KUKA KRL program: MyProgram_239().src

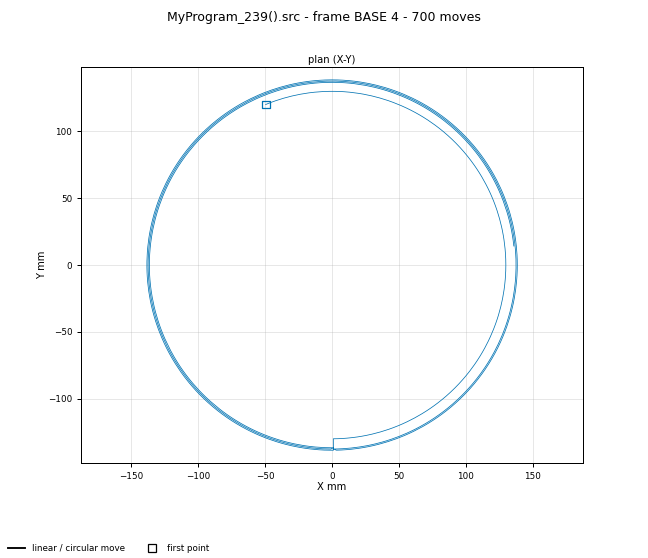
[picture p0: tool path of MyProgram_239().src in frame BASE 4, 700 of 700 moves have a stored position in this frame; points joined in program order, loops and branches not executed]
&ACCESS RVP
&REL 1
&PARAM TEMPLATE = C:\KRC\Roboter\Template\vorgabe
&PARAM EDITMASK = *
DEF MyProgram_239()
; ---- Setting reference (Base) ----
$BASE = BASE_DATA[4]

; --------------------------
; ---- Setting tool (TCP) ----
$TOOL = TOOL_DATA[3]
; --------------------------

$VEL.CP = VEL_APROX_PRINT
Startdeposition()
$VEL.CP = VEL_PRINT
LIN {X -49.7032,Y 120.0061,Z 160,A 111.2749,B 14.0881,C -0.1993,E1 14.0298,E2 338.4805} C_DIS
LIN {X -45.6946,Y 121.5885,Z 160,A 109.4151,B 14.0881,C -0.2026,E1 14.0346,E2 340.334} C_DIS
LIN {X -42.2336,Y 122.834,Z 160,A 107.7853,B 14.0881,C -0.2041,E1 14.0389,E2 341.9633} C_DIS
LIN {X -39.2151,Y 123.8307,Z 160,A 106.3787,B 14.0881,C -0.2054,E1 14.0427,E2 343.3693} C_DIS
LIN {X -36.1716,Y 124.7537,Z 160,A 104.9717,B 14.088,C -0.2066,E1 14.0464,E2 344.7756} C_DIS
LIN {X -33.1062,Y 125.6021,Z 160,A 103.5625,B 14.088,C -0.2076,E1 14.0502,E2 346.1844} C_DIS
LIN {X -29.9974,Y 126.381,Z 160,A 102.1496,B 14.088,C -0.2088,E1 14.0541,E2 347.5962} C_DIS
LIN {X -26.9022,Y 127.0761,Z 160,A 100.7679,B 14.088,C -0.2103,E1 14.0578,E2 348.9749} C_DIS
LIN {X -23.6832,Y 127.7162,Z 160,A 99.3021,B 14.088,C -0.2107,E1 14.0618,E2 350.4419} C_DIS
LIN {X -21.0729,Y 128.1711,Z 160,A 98.0756,B 14.088,C -0.2098,E1 14.0652,E2 351.6741} C_DIS
LIN {X -17.5361,Y 128.7041,Z 160,A 96.3923,B 14.088,C -0.2077,E1 14.0699,E2 353.3685} C_DIS
LIN {X -13.1972,Y 129.2214,Z 160,A 94.4723,B 14.088,C -0.2087,E1 14.0752,E2 355.2865} C_DIS
LIN {X -9.5576,Y 129.5396,Z 160,A 92.993,B 14.088,C -0.2129,E1 14.0793,E2 356.7497} C_DIS
LIN {X -6.3664,Y 129.7357,Z 160,A 91.5337,B 14.088,C -0.2119,E1 14.0834,E2 358.2139} C_DIS
LIN {X -2.0579,Y 129.8755,Z 160,A 89.6356,B 14.088,C -0.2123,E1 14.0887,E2 360.1106} C_DIS
LIN {X 2.062,Y 129.8755,Z 160,A 87.7741,B 14.088,C -0.2112,E1 14.0939,E2 361.9764} C_DIS
LIN {X 5.2462,Y 129.7859,Z 160,A 86.3414,B 14.088,C -0.2104,E1 14.0979,E2 363.4116} C_DIS
LIN {X 9.0939,Y 129.5735,Z 160,A 84.7482,B 14.0879,C -0.2132,E1 14.1023,E2 364.9919} C_DIS
LIN {X 13.1987,Y 129.2212,Z 160,A 82.7681,B 14.0879,C -0.2083,E1 14.1079,E2 366.9899} C_DIS
LIN {X 17.4787,Y 128.7116,Z 160,A 81.0931,B 14.0879,C -0.2141,E1 14.1124,E2 368.6386} C_DIS
LIN {X 20.1102,Y 128.3256,Z 160,A 79.7906,B 14.0879,C -0.21,E1 14.1161,E2 369.9554} C_DIS
LIN {X 23.3548,Y 127.7755,Z 160,A 78.4283,B 14.0879,C -0.2119,E1 14.1198,E2 371.3071} C_DIS
LIN {X 26.9191,Y 127.0724,Z 160,A 76.937,B 14.0879,C -0.2142,E1 14.1238,E2 372.7854} C_DIS
LIN {X 29.569,Y 126.4828,Z 160,A 75.6327,B 14.0879,C -0.2105,E1 14.1274,E2 374.1017} C_DIS
LIN {X 32.6519,Y 125.7225,Z 160,A 74.2354,B 14.0879,C -0.2097,E1 14.1312,E2 375.4984} C_DIS
LIN {X 35.7407,Y 124.8799,Z 160,A 72.8179,B 14.0879,C -0.2085,E1 14.135,E2 376.9163} C_DIS
LIN {X 38.7913,Y 123.9661,Z 160,A 71.4198,B 14.0879,C -0.2076,E1 14.1387,E2 378.3136} C_DIS
LIN {X 41.8166,Y 122.9786,Z 160,A 69.7915,B 14.0881,C -0.1999,E1 14.1431,E2 379.9674} C_DIS
LIN {X 45.6939,Y 121.5888,Z 160,A 68.1327,B 14.0881,C -0.2027,E1 14.1474,E2 381.608} C_DIS
LIN {X 49.2665,Y 120.1879,Z 160,A 66.5276,B 14.0881,C -0.2035,E1 14.1516,E2 383.2031} C_DIS
LIN {X 51.7426,Y 119.1406,Z 160,A 65.2806,B 14.0881,C -0.2004,E1 14.1548,E2 384.4571} C_DIS
LIN {X 55.5451,Y 117.4168,Z 160,A 63.5143,B 14.0881,C -0.2004,E1 14.1592,E2 386.2149} C_DIS
LIN {X 58.8237,Y 115.8081,Z 160,A 61.8469,B 14.0881,C -0.1968,E1 14.1634,E2 387.8889} C_DIS
LIN {X 62.2203,Y 114.0214,Z 160,A 60.1436,B 14.0881,C -0.1942,E1 14.1676,E2 389.5937} C_DIS
LIN {X 65.3999,Y 112.2284,Z 160,A 58.6138,B 14.0881,C -0.1942,E1 14.1713,E2 391.1146} C_DIS
LIN {X 68.1296,Y 110.5923,Z 160,A 57.1082,B 14.0882,C -0.1892,E1 14.1749,E2 392.6322} C_DIS
LIN {X 71.7854,Y 108.2555,Z 160,A 55.3158,B 14.0882,C -0.1898,E1 14.1791,E2 394.4111} C_DIS
LIN {X 74.4134,Y 106.4657,Z 160,A 53.9209,B 14.0882,C -0.1878,E1 14.1823,E2 395.8055} C_DIS
LIN {X 77.0015,Y 104.6089,Z 160,A 52.4462,B 14.0883,C -0.1833,E1 14.1856,E2 397.2886} C_DIS
LIN {X 80.232,Y 102.1521,Z 160,A 50.645,B 14.0883,C -0.1798,E1 14.1896,E2 399.0918} C_DIS
LIN {X 83.2585,Y 99.7013,Z 160,A 48.9085,B 14.0884,C -0.1761,E1 14.1934,E2 400.8311} C_DIS
LIN {X 86.6409,Y 96.7759,Z 160,A 46.989,B 14.0884,C -0.174,E1 14.1974,E2 402.7452} C_DIS
LIN {X 89.734,Y 93.9151,Z 160,A 45.1415,B 14.0884,C -0.1706,E1 14.2012,E2 404.5923} C_DIS
LIN {X 92.613,Y 91.0774,Z 160,A 43.3362,B 14.0885,C -0.1663,E1 14.2047,E2 406.4011} C_DIS
LIN {X 95.7938,Y 87.7259,Z 160,A 41.3052,B 14.0885,C -0.1622,E1 14.2086,E2 408.4323} C_DIS
LIN {X 98.5161,Y 84.6572,Z 160,A 39.5451,B 14.0885,C -0.1597,E1 14.2118,E2 410.1878} C_DIS
LIN {X 101.2684,Y 81.345,Z 160,A 37.6742,B 14.0886,C -0.1563,E1 14.2151,E2 412.0566} C_DIS
LIN {X 103.9483,Y 77.8918,Z 160,A 35.7201,B 14.0886,C -0.151,E1 14.2184,E2 414.0149} C_DIS
LIN {X 106.1955,Y 74.7981,Z 160,A 34.1837,B 14.0886,C -0.1516,E1 14.2209,E2 415.535} C_DIS
LIN {X 107.9969,Y 72.1728,Z 160,A 32.7951,B 14.0887,C -0.1487,E1 14.2231,E2 416.9228} C_DIS
LIN {X 109.9996,Y 69.0825,Z 160,A 31.0479,B 14.0887,C -0.1409,E1 14.2257,E2 418.6855} C_DIS
LIN {X 111.9911,Y 65.8044,Z 160,A 29.5076,B 14.0887,C -0.1413,E1 14.2279,E2 420.2095} C_DIS
LIN {X 113.5692,Y 63.0419,Z 160,A 28.0941,B 14.0888,C -0.1374,E1 14.2299,E2 421.6253} C_DIS
LIN {X 115.0779,Y 60.2396,Z 160,A 26.7243,B 14.0888,C -0.1348,E1 14.2316,E2 422.9922} C_DIS
LIN {X 116.5193,Y 57.402,Z 160,A 25.3351,B 14.0888,C -0.1316,E1 14.2334,E2 424.3809} C_DIS
LIN {X 118.088,Y 54.1033,Z 160,A 23.7352,B 14.0889,C -0.1276,E1 14.2353,E2 425.981} C_DIS
LIN {X 119.3878,Y 51.1708,Z 160,A 22.3362,B 14.0889,C -0.1243,E1 14.2368,E2 427.3793} C_DIS
LIN {X 120.7817,Y 47.7926,Z 160,A 20.6564,B 14.0889,C -0.1177,E1 14.2386,E2 429.0686} C_DIS
LIN {X 122.1392,Y 44.2018,Z 160,A 18.978,B 14.089,C -0.1135,E1 14.2402,E2 430.7468} C_DIS
LIN {X 123.3413,Y 40.7281,Z 160,A 17.4623,B 14.089,C -0.1123,E1 14.2416,E2 432.2517} C_DIS
LIN {X 124.3013,Y 37.697,Z 160,A 16.0749,B 14.089,C -0.1088,E1 14.2427,E2 433.6387} C_DIS
LIN {X 125.187,Y 34.6425,Z 160,A 14.6877,B 14.089,C -0.1052,E1 14.2438,E2 435.0256} C_DIS
LIN {X 125.9978,Y 31.5675,Z 160,A 13.3007,B 14.0891,C -0.1017,E1 14.2447,E2 436.4121} C_DIS
LIN {X 126.7327,Y 28.4748,Z 160,A 11.9153,B 14.0891,C -0.0982,E1 14.2456,E2 437.7971} C_DIS
LIN {X 127.2976,Y 25.829,Z 160,A 10.7066,B 14.0891,C -0.0942,E1 14.2463,E2 439.0088} C_DIS
LIN {X 127.9907,Y 22.1528,Z 160,A 9.1132,B 14.0891,C -0.0911,E1 14.2471,E2 440.5974} C_DIS
LIN {X 128.4876,Y 19.0587,Z 160,A 7.716,B 14.0892,C -0.0866,E1 14.2477,E2 441.9979} C_DIS
LIN {X 128.9711,Y 15.4368,Z 160,A 6.049,B 14.0892,C -0.0801,E1 14.2483,E2 443.6731} C_DIS
LIN {X 129.3109,Y 12.2699,Z 160,A 4.6342,B 14.0892,C -0.0756,E1 14.2487,E2 445.0907} C_DIS
LIN {X 129.6473,Y 7.9637,Z 160,A 2.8627,B 14.0892,C -0.0741,E1 14.249,E2 446.8487} C_DIS
LIN {X 129.822,Y 4.3136,Z 160,A 1.0954,B 14.0893,C -0.0644,E1 14.2492,E2 448.636} C_DIS
LIN {X 129.895,Y 0.007,Z 160,A -0.785,B 14.0893,C -0.0593,E1 14.2492,E2 450.5165} C_DIS
LIN {X 129.822,Y -4.3151,Z 160,A -2.4696,B 14.0893,C -0.0606,E1 14.2492,E2 452.1773} C_DIS
LIN {X 129.676,Y -7.498,Z 160,A -3.9032,B 14.0893,C -0.0555,E1 14.249,E2 453.6158} C_DIS
LIN {X 129.4525,Y -10.6747,Z 160,A -5.4288,B 14.0894,C -0.0475,E1 14.2486,E2 455.1574} C_DIS
LIN {X 128.9724,Y -15.4254,Z 160,A -7.4213,B 14.0894,C -0.0448,E1 14.248,E2 457.1391} C_DIS
LIN {X 128.5535,Y -18.5974,Z 160,A -8.7549,B 14.0894,C -0.043,E1 14.2475,E2 458.4653} C_DIS
LIN {X 127.9752,Y -22.2393,Z 160,A -10.3122,B 14.0894,C -0.0403,E1 14.2468,E2 460.0166} C_DIS
LIN {X 127.4877,Y -24.8786,Z 160,A -11.6353,B 14.0894,C -0.0324,E1 14.2461,E2 461.3574} C_DIS
LIN {X 126.8347,Y -28.0205,Z 160,A -12.933,B 14.0894,C -0.0319,E1 14.2454,E2 462.6432} C_DIS
LIN {X 126.1505,Y -30.9533,Z 160,A -14.2383,B 14.0894,C -0.0288,E1 14.2445,E2 463.9474} C_DIS
LIN {X 125.3166,Y -34.1769,Z 160,A -15.7036,B 14.0894,C -0.0246,E1 14.2435,E2 465.4142} C_DIS
LIN {X 124.433,Y -37.2667,Z 160,A -17.1097,B 14.0894,C -0.0208,E1 14.2424,E2 466.8207} C_DIS
LIN {X 123.4826,Y -40.3039,Z 160,A -18.4978,B 14.0894,C -0.0172,E1 14.2412,E2 468.2088} C_DIS
LIN {X 122.2991,Y -43.7581,Z 160,A -20.2163,B 14.0894,C -0.0092,E1 14.2396,E2 469.942} C_DIS
LIN {X 120.7401,Y -47.8966,Z 160,A -22.0062,B 14.0894,C -0.0087,E1 14.2378,E2 471.7155} C_DIS
LIN {X 119.5532,Y -50.7878,Z 160,A -23.3927,B 14.0894,C -0.0046,E1 14.2363,E2 473.1047} C_DIS
LIN {X 118.3107,Y -53.6163,Z 160,A -24.7448,B 14.0894,C -0.0011,E1 14.2348,E2 474.4573} C_DIS
LIN {X 116.7283,Y -56.9782,Z 160,A -26.352,B 14.0894,C 0.0024,E1 14.2328,E2 476.0628} C_DIS
LIN {X 115.2981,Y -59.8203,Z 160,A -27.7239,B 14.0894,C 0.0053,E1 14.2311,E2 477.4328} C_DIS
LIN {X 114.1159,Y -62.047,Z 160,A -28.9697,B 14.0894,C 0.0125,E1 14.2294,E2 478.6958} C_DIS
LIN {X 112.4647,Y -64.9918,Z 160,A -30.4091,B 14.0894,C 0.0149,E1 14.2274,E2 480.1312} C_DIS
LIN {X 110.5875,Y -68.1374,Z 160,A -31.9279,B 14.0894,C 0.0161,E1 14.2252,E2 481.6406} C_DIS
LIN {X 108.5876,Y -71.2811,Z 160,A -33.662,B 14.0894,C 0.0232,E1 14.2226,E2 483.3874} C_DIS
LIN {X 106.4641,Y -74.4157,Z 160,A -35.2113,B 14.0894,C 0.0237,E1 14.2202,E2 484.9246} C_DIS
LIN {X 104.6112,Y -76.9983,Z 160,A -36.5974,B 14.0894,C 0.0267,E1 14.2179,E2 486.3106} C_DIS
LIN {X 102.8556,Y -79.3288,Z 160,A -38.0201,B 14.0894,C 0.0341,E1 14.2155,E2 487.7509} C_DIS
LIN {X 100.2422,Y -82.6064,Z 160,A -39.8187,B 14.0894,C 0.037,E1 14.2123,E2 489.5459} C_DIS
LIN {X 97.4592,Y -85.8719,Z 160,A -41.6299,B 14.0894,C 0.039,E1 14.209,E2 491.3497} C_DIS
LIN {X 94.7928,Y -88.8071,Z 160,A -43.3846,B 14.0894,C 0.0431,E1 14.2057,E2 493.1072} C_DIS
LIN {X 91.8229,Y -91.8745,Z 160,A -45.341,B 14.0894,C 0.0496,E1 14.2018,E2 495.0744} C_DIS
LIN {X 88.5345,Y -95.0467,Z 160,A -47.2615,B 14.0894,C 0.0511,E1 14.198,E2 496.9861} C_DIS
LIN {X 85.452,Y -97.8273,Z 160,A -49.0529,B 14.0894,C 0.0537,E1 14.1942,E2 498.7749} C_DIS
LIN {X 82.3877,Y -100.4219,Z 160,A -50.8685,B 14.0894,C 0.0586,E1 14.1903,E2 500.5977} C_DIS
LIN {X 79.231,Y -102.9313,Z 160,A -52.6764,B 14.0894,C 0.063,E1 14.1863,E2 502.4111} C_DIS
LIN {X 76.4378,Y -105.0217,Z 160,A -54.1414,B 14.0894,C 0.0637,E1 14.183,E2 503.869} C_DIS
LIN {X 73.4926,Y -107.1031,Z 160,A -55.6315,B 14.0894,C 0.0635,E1 14.1796,E2 505.3489} C_DIS
LIN {X 70.8271,Y -108.8842,Z 160,A -57.1232,B 14.0894,C 0.0684,E1 14.1761,E2 506.8514} C_DIS
LIN {X 67.1774,Y -111.173,Z 160,A -58.9257,B 14.0894,C 0.0686,E1 14.1719,E2 508.6442} C_DIS
LIN {X 64.4349,Y -112.7847,Z 160,A -60.3238,B 14.0894,C 0.0708,E1 14.1685,E2 510.0432} C_DIS
LIN {X 61.7406,Y -114.2822,Z 160,A -61.7623,B 14.0893,C 0.0753,E1 14.165,E2 511.4923} C_DIS
LIN {X 58.8215,Y -115.8091,Z 160,A -63.1186,B 14.0893,C 0.0745,E1 14.1616,E2 512.8385} C_DIS
LIN {X 55.9699,Y -117.2139,Z 160,A -64.5849,B 14.0893,C 0.0785,E1 14.1579,E2 514.3138} C_DIS
LIN {X 52.6245,Y -118.7543,Z 160,A -66.1324,B 14.0893,C 0.0784,E1 14.154,E2 515.8537} C_DIS
LIN {X 49.6988,Y -120.008,Z 160,A -67.5761,B 14.0893,C 0.0814,E1 14.1503,E2 517.3034} C_DIS
LIN {X 45.6909,Y -121.5899,Z 160,A -69.4181,B 14.0893,C 0.082,E1 14.1455,E2 519.1401} C_DIS
LIN {X 42.2559,Y -122.8263,Z 160,A -71.0351,B 14.0893,C 0.084,E1 14.1412,E2 520.7593} C_DIS
LIN {X 39.1603,Y -123.8482,Z 160,A -72.4527,B 14.0893,C 0.0849,E1 14.1374,E2 522.1757} C_DIS
LIN {X 36.1394,Y -124.7632,Z 160,A -73.8392,B 14.0893,C 0.0861,E1 14.1337,E2 523.5625} C_DIS
LIN {X 33.0912,Y -125.6061,Z 160,A -75.2287,B 14.0893,C 0.0873,E1 14.13,E2 524.9525} C_DIS
LIN {X 30.02,Y -126.3755,Z 160,A -76.6903,B 14.0892,C 0.0904,E1 14.126,E2 526.4228} C_DIS
LIN {X 25.8513,Y -127.293,Z 160,A -78.5312,B 14.0892,C 0.0906,E1 14.121,E2 528.2601} C_DIS
LIN {X 22.2073,Y -127.9809,Z 160,A -80.1101,B 14.0892,C 0.0901,E1 14.1167,E2 529.8335} C_DIS
LIN {X 19.0624,Y -128.4871,Z 160,A -81.5115,B 14.0892,C 0.0908,E1 14.1128,E2 531.2354} C_DIS
LIN {X 15.4256,Y -128.9724,Z 160,A -83.2363,B 14.0892,C 0.0947,E1 14.108,E2 532.9737} C_DIS
LIN {X 11.1426,Y -129.413,Z 160,A -85.052,B 14.0892,C 0.0932,E1 14.103,E2 534.7807} C_DIS
LIN {X 7.9646,Y -129.6473,Z 160,A -86.4484,B 14.0892,C 0.0934,E1 14.0991,E2 536.1768} C_DIS
LIN {X 4.2979,Y -129.8225,Z 160,A -88.2381,B 14.0892,C 0.0987,E1 14.094,E2 537.9875} C_DIS
LIN {X 0.9217,Y -129.8856,Z 160,A -89.155,B 14.0892,C 0.0825,E1 14.0916,E2 538.8374} C_DIS
Enddeposition()
LIN {X 0.9743,Y -138.4568,Z 161,A -92.8969,B 24.9726,C -1.2087,E1 25.0002,E2 539.6734} C_DIS
Startdeposition()
$VEL.CP = VEL_PRINT
LIN {X -3.1683,Y -138.4258,Z 161,A -94.4704,B 24.9723,C -1.216,E1 24.9959,E2 541.2295} C_DIS
LIN {X -5.6886,Y -138.3438,Z 161,A -95.6511,B 24.9727,C -1.2084,E1 24.9925,E2 542.4283} C_DIS
LIN {X -10.1591,Y -138.0871,Z 161,A -97.4064,B 24.9724,C -1.2137,E1 24.9877,E2 544.1717} C_DIS
LIN {X -13.2488,Y -137.825,Z 161,A -98.6993,B 24.9724,C -1.2133,E1 24.9841,E2 545.4663} C_DIS
LIN {X -16.4453,Y -137.4802,Z 161,A -100.0746,B 24.9725,C -1.211,E1 24.9802,E2 546.8479} C_DIS
LIN {X -20.7998,Y -136.8895,Z 161,A -101.9215,B 24.9725,C -1.2099,E1 24.9751,E2 548.6988} C_DIS
LIN {X -24.7621,Y -136.2285,Z 161,A -103.6222,B 24.9727,C -1.2084,E1 24.9704,E2 550.4048} C_DIS
LIN {X -30.0439,Y -135.1637,Z 161,A -105.7422,B 24.9723,C -1.2153,E1 24.9647,E2 552.511} C_DIS
LIN {X -34.7423,Y -134.0323,Z 161,A -107.7572,B 24.9723,C -1.2156,E1 24.9592,E2 554.528} C_DIS
LIN {X -38.0185,Y -133.1403,Z 161,A -109.1637,B 24.9723,C -1.2165,E1 24.9554,E2 555.9347} C_DIS
LIN {X -41.2654,Y -132.1701,Z 161,A -110.5701,B 24.9723,C -1.2173,E1 24.9517,E2 557.3415} C_DIS
LIN {X -44.4935,Y -131.1187,Z 161,A -111.9792,B 24.9723,C -1.2183,E1 24.9479,E2 558.751} C_DIS
LIN {X -47.085,Y -130.2082,Z 161,A -113.175,B 24.9723,C -1.2162,E1 24.9448,E2 559.9543} C_DIS
LIN {X -50.5394,Y -128.9072,Z 161,A -114.7424,B 24.9723,C -1.2155,E1 24.9407,E2 561.5265} C_DIS
LIN {X -54.2078,Y -127.41,Z 161,A -116.2763,B 24.972,C -1.2229,E1 24.9367,E2 563.0464} C_DIS
LIN {X -57.1309,Y -126.1254,Z 161,A -117.75,B 24.9723,C -1.2163,E1 24.9329,E2 564.5393} C_DIS
LIN {X -61.082,Y -124.2584,Z 161,A -119.4559,B 24.9719,C -1.224,E1 24.9287,E2 566.2313} C_DIS
LIN {X -64.4095,Y -122.5665,Z 161,A -120.964,B 24.9718,C -1.228,E1 24.925,E2 567.7341} C_DIS
LIN {X -67.5702,Y -120.8555,Z 161,A -122.6011,B 24.972,C -1.2221,E1 24.9209,E2 569.3898} C_DIS
LIN {X -71.6995,Y -118.4519,Z 161,A -124.5871,B 24.972,C -1.2246,E1 24.9161,E2 571.376} C_DIS
LIN {X -75.1902,Y -116.2676,Z 161,A -126.1567,B 24.9715,C -1.2343,E1 24.9125,E2 572.9274} C_DIS
LIN {X -78.5445,Y -114.0285,Z 161,A -127.9061,B 24.9715,C -1.2329,E1 24.9084,E2 574.686} C_DIS
LIN {X -82.2199,Y -111.4076,Z 161,A -129.8161,B 24.9715,C -1.234,E1 24.9041,E2 576.6001} C_DIS
LIN {X -85.6942,Y -108.7576,Z 161,A -131.6209,B 24.9713,C -1.2375,E1 24.9001,E2 578.4031} C_DIS
LIN {X -89.11,Y -105.9769,Z 161,A -133.4578,B 24.9712,C -1.2403,E1 24.8962,E2 580.2403} C_DIS
LIN {X -92.5782,Y -102.9613,Z 161,A -135.2743,B 24.9708,C -1.2486,E1 24.8924,E2 582.0443} C_DIS
LIN {X -95.3764,Y -100.3751,Z 161,A -136.9551,B 24.9709,C -1.2465,E1 24.8889,E2 583.737} C_DIS
LIN {X -98.5504,Y -97.2609,Z 161,A -138.8238,B 24.9708,C -1.249,E1 24.8852,E2 585.6075} C_DIS
LIN {X -101.7004,Y -93.9618,Z 161,A -140.6893,B 24.9705,C -1.2545,E1 24.8817,E2 587.4683} C_DIS
LIN {X -104.6037,Y -90.7189,Z 161,A -142.4757,B 24.9703,C -1.2594,E1 24.8784,E2 589.2509} C_DIS
LIN {X -107.3011,Y -87.5109,Z 161,A -144.286,B 24.9703,C -1.2597,E1 24.8751,E2 591.0689} C_DIS
LIN {X -110.316,Y -83.679,Z 161,A -146.1965,B 24.9698,C -1.2703,E1 24.8719,E2 592.9634} C_DIS
LIN {X -112.9457,Y -80.0941,Z 161,A -148.1613,B 24.9698,C -1.2685,E1 24.8687,E2 594.9419} C_DIS
LIN {X -115.6061,Y -76.203,Z 161,A -149.7905,B 24.9688,C -1.2902,E1 24.8662,E2 596.5275} C_DIS
LIN {X -117.2158,Y -73.7034,Z 161,A -151.3483,B 24.9695,C -1.2767,E1 24.8638,E2 598.1255} C_DIS
LIN {X -119.4368,Y -70.0467,Z 161,A -153.1361,B 24.9693,C -1.2806,E1 24.8612,E2 599.9131} C_DIS
LIN {X -121.715,Y -66.0095,Z 161,A -155.0718,B 24.9691,C -1.2851,E1 24.8586,E2 601.8484} C_DIS
LIN {X -123.774,Y -62.0629,Z 161,A -156.7926,B 24.9685,C -1.2965,E1 24.8564,E2 603.5511} C_DIS
LIN {X -125.4195,Y -58.6639,Z 161,A -158.5603,B 24.9688,C -1.2906,E1 24.8543,E2 605.3425} C_DIS
LIN {X -127.3665,Y -54.3084,Z 161,A -160.3524,B 24.9681,C -1.3057,E1 24.8523,E2 607.1084} C_DIS
LIN {X -128.6643,Y -51.1573,Z 161,A -161.7697,B 24.9679,C -1.3096,E1 24.8508,E2 608.5244} C_DIS
LIN {X -129.8581,Y -48.0452,Z 161,A -163.1325,B 24.9676,C -1.3146,E1 24.8495,E2 609.883} C_DIS
LIN {X -131.9081,Y -42.0882,Z 161,A -166.3797,B 24.9688,C -1.2903,E1 24.8466,E2 613.2067} C_DIS
LIN {X -133.326,Y -37.3544,Z 161,A -167.8163,B 24.967,C -1.3274,E1 24.8455,E2 614.5632} C_DIS
LIN {X -134.165,Y -34.2194,Z 161,A -169.2421,B 24.967,C -1.3274,E1 24.8445,E2 615.9973} C_DIS
LIN {X -135.1015,Y -30.316,Z 161,A -170.8508,B 24.9666,C -1.3353,E1 24.8435,E2 617.5965} C_DIS
LIN {X -135.9103,Y -26.454,Z 161,A -172.5696,B 24.9666,C -1.3362,E1 24.8425,E2 619.3234} C_DIS
LIN {X -136.5611,Y -22.8535,Z 161,A -174.0223,B 24.9662,C -1.3442,E1 24.8418,E2 620.7656} C_DIS
LIN {X -137.0663,Y -19.5976,Z 161,A -175.401,B 24.966,C -1.3479,E1 24.8413,E2 622.1438} C_DIS
LIN {X -137.5029,Y -16.255,Z 161,A -176.7899,B 24.9657,C -1.3528,E1 24.8408,E2 623.5294} C_DIS
LIN {X -137.8589,Y -12.8957,Z 161,A -178.3316,B 24.9659,C -1.3501,E1 24.8404,E2 625.0867} C_DIS
LIN {X -138.1811,Y -8.7939,Z 161,A -179.9255,B 24.9653,C -1.3612,E1 24.8401,E2 626.6638} C_DIS
LIN {X -138.353,Y -5.4532,Z 161,A 178.6682,B 24.9651,C -1.3646,E1 24.8399,E2 628.0703} C_DIS
LIN {X -138.4547,Y -1.4284,Z 161,A 176.8431,B 24.9652,C -1.3621,E1 24.8398,E2 629.9125} C_DIS
LIN {X -138.4329,Y 2.8047,Z 161,A 175.2532,B 24.9645,C -1.3761,E1 24.8398,E2 631.4786} C_DIS
LIN {X -138.3232,Y 6.2058,Z 161,A 173.8012,B 24.9645,C -1.3785,E1 24.84,E2 632.9335} C_DIS
LIN {X -138.1334,Y 9.5261,Z 161,A 172.3092,B 24.9645,C -1.3773,E1 24.8403,E2 634.4374} C_DIS
LIN {X -137.7951,Y 13.5601,Z 161,A 170.7533,B 24.9639,C -1.3889,E1 24.8407,E2 635.975} C_DIS
LIN {X -137.423,Y 16.9246,Z 161,A 169.3455,B 24.9636,C -1.3932,E1 24.8411,E2 637.3811} C_DIS
LIN {X -136.971,Y 20.2641,Z 161,A 167.9566,B 24.9634,C -1.3981,E1 24.8416,E2 638.7666} C_DIS
LIN {X -136.45,Y 23.5193,Z 161,A 166.4063,B 24.9636,C -1.3932,E1 24.8424,E2 640.3377} C_DIS
LIN {X -135.5939,Y 28.0303,Z 161,A 164.5764,B 24.9631,C -1.403,E1 24.8434,E2 642.1551} C_DIS
LIN {X -134.7645,Y 31.7835,Z 161,A 163.0674,B 24.9626,C -1.4123,E1 24.8443,E2 643.6508} C_DIS
LIN {X -133.978,Y 34.9525,Z 161,A 161.7054,B 24.9624,C -1.4162,E1 24.8452,E2 645.0115} C_DIS
LIN {X -133.1336,Y 38.0424,Z 161,A 160.3415,B 24.9624,C -1.4185,E1 24.8462,E2 646.3776} C_DIS
LIN {X -132.1906,Y 41.1986,Z 161,A 158.974,B 24.9621,C -1.4227,E1 24.8474,E2 647.7431} C_DIS
LIN {X -131.2402,Y 44.1287,Z 161,A 157.7051,B 24.9618,C -1.4271,E1 24.8485,E2 649.0087} C_DIS
LIN {X -130.0732,Y 47.4594,Z 161,A 156.2083,B 24.9617,C -1.43,E1 24.8499,E2 650.5072} C_DIS
LIN {X -128.5676,Y 51.3973,Z 161,A 154.3548,B 24.9617,C -1.43,E1 24.8518,E2 652.371} C_DIS
LIN {X -126.9828,Y 55.1959,Z 161,A 152.7439,B 24.9612,C -1.44,E1 24.8535,E2 653.9671} C_DIS
LIN {X -125.6195,Y 58.2312,Z 161,A 151.3722,B 24.9609,C -1.4445,E1 24.8551,E2 655.3354} C_DIS
LIN {X -124.2449,Y 61.1094,Z 161,A 149.9388,B 24.961,C -1.4429,E1 24.8569,E2 656.7806} C_DIS
LIN {X -122.1777,Y 65.1497,Z 161,A 148.1497,B 24.9604,C -1.453,E1 24.8591,E2 658.555} C_DIS
LIN {X -120.2763,Y 68.595,Z 161,A 146.4555,B 24.9604,C -1.4546,E1 24.8615,E2 660.2545} C_DIS
LIN {X -118.2785,Y 71.9863,Z 161,A 144.7299,B 24.9604,C -1.4545,E1 24.8639,E2 661.9892} C_DIS
LIN {X -115.745,Y 75.9921,Z 161,A 142.8285,B 24.9599,C -1.4632,E1 24.8668,E2 663.8795} C_DIS
LIN {X -113.4997,Y 79.3067,Z 161,A 141.2587,B 24.9594,C -1.4723,E1 24.8693,E2 665.4352} C_DIS
LIN {X -111.2951,Y 82.3725,Z 161,A 139.5237,B 24.9596,C -1.4679,E1 24.8721,E2 667.1891} C_DIS
LIN {X -108.437,Y 86.0995,Z 161,A 137.5624,B 24.9594,C -1.4724,E1 24.8755,E2 669.1492} C_DIS
LIN {X -105.4296,Y 89.7568,Z 161,A 135.5991,B 24.9591,C -1.4774,E1 24.879,E2 671.1094} C_DIS
LIN {X -102.6916,Y 92.8771,Z 161,A 133.8802,B 24.9589,C -1.4818,E1 24.8822,E2 672.8256} C_DIS
LIN {X -99.8708,Y 95.9042,Z 161,A 132.1529,B 24.9587,C -1.4854,E1 24.8855,E2 674.5518} C_DIS
LIN {X -96.8928,Y 98.9114,Z 161,A 130.3843,B 24.9585,C -1.4889,E1 24.889,E2 676.3196} C_DIS
LIN {X -93.8532,Y 101.8003,Z 161,A 128.6555,B 24.9582,C -1.4934,E1 24.8926,E2 678.0448} C_DIS
LIN {X -90.7611,Y 104.5668,Z 161,A 126.9095,B 24.9581,C -1.4959,E1 24.8962,E2 679.7917} C_DIS
LIN {X -87.0746,Y 107.6556,Z 161,A 125.0068,B 24.9576,C -1.5049,E1 24.9003,E2 681.6802} C_DIS
LIN {X -83.6906,Y 110.3072,Z 161,A 123.1274,B 24.9576,C -1.5036,E1 24.9045,E2 683.5694} C_DIS
LIN {X -79.8229,Y 113.137,Z 161,A 121.1414,B 24.9574,C -1.5077,E1 24.909,E2 685.5528} C_DIS
LIN {X -75.8058,Y 115.8677,Z 161,A 119.237,B 24.9569,C -1.5171,E1 24.9133,E2 687.441} C_DIS
LIN {X -72.4221,Y 118.0115,Z 161,A 117.5953,B 24.9566,C -1.5211,E1 24.9172,E2 689.0783} C_DIS
LIN {X -68.9984,Y 120.0462,Z 161,A 115.8797,B 24.9566,C -1.5207,E1 24.9214,E2 690.8002} C_DIS
LIN {X -65.4381,Y 122.0227,Z 161,A 113.9576,B 24.9572,C -1.5114,E1 24.9261,E2 692.7498} C_DIS
LIN {X -60.7957,Y 124.3996,Z 161,A 112.0075,B 24.9564,C -1.5258,E1 24.9309,E2 694.6709} C_DIS
LIN {X -57.3003,Y 126.0497,Z 161,A 110.4633,B 24.9561,C -1.5311,E1 24.9348,E2 696.2063} C_DIS
LIN {X -54.6355,Y 127.2251,Z 161,A 109.2314,B 24.9561,C -1.5316,E1 24.938,E2 697.44} C_DIS
LIN {X -51.4595,Y 128.5425,Z 161,A 107.787,B 24.956,C -1.5325,E1 24.9417,E2 698.8854} C_DIS
LIN {X -48.0831,Y 129.8439,Z 161,A 106.3544,B 24.9557,C -1.5379,E1 24.9454,E2 700.3081} C_DIS
LIN {X -45.3398,Y 130.8261,Z 161,A 105.161,B 24.9556,C -1.5401,E1 24.9486,E2 701.4986} C_DIS
LIN {X -41.8358,Y 131.9887,Z 161,A 103.606,B 24.9556,C -1.5406,E1 24.9527,E2 703.0555} C_DIS
LIN {X -38.8437,Y 132.8998,Z 161,A 102.2741,B 24.9556,C -1.5401,E1 24.9563,E2 704.3908} C_DIS
LIN {X -35.5522,Y 133.818,Z 161,A 100.8733,B 24.9554,C -1.5423,E1 24.9601,E2 705.7886} C_DIS
LIN {X -32.2798,Y 134.6448,Z 161,A 99.4741,B 24.9554,C -1.5435,E1 24.9638,E2 707.1868} C_DIS
LIN {X -28.9921,Y 135.391,Z 161,A 98.0849,B 24.9553,C -1.5451,E1 24.9676,E2 708.574} C_DIS
LIN {X -25.6499,Y 136.064,Z 161,A 96.6746,B 24.9553,C -1.5463,E1 24.9715,E2 709.983} C_DIS
LIN {X -21.6008,Y 136.7655,Z 161,A 94.9369,B 24.9553,C -1.5455,E1 24.9763,E2 711.7241} C_DIS
LIN {X -17.8049,Y 137.3108,Z 161,A 92.9784,B 24.9563,C -1.5269,E1 24.9818,E2 713.7282} C_DIS
LIN {X -13.8852,Y 137.7639,Z 161,A 91.5053,B 24.9558,C -1.5362,E1 24.9859,E2 715.1801} C_DIS
LIN {X -9.5521,Y 138.1315,Z 161,A 89.8147,B 24.9554,C -1.5428,E1 24.9905,E2 716.8558} C_DIS
LIN {X -5.2372,Y 138.3614,Z 161,A 88.1896,B 24.9549,C -1.5521,E1 24.995,E2 718.4592} C_DIS
LIN {X -0.3944,Y 138.4604,Z 161,A 85.985,B 24.9555,C -1.5419,E1 25.0012,E2 720.6881} C_DIS
LIN {X 4.1453,Y 138.3986,Z 161,A 84.2451,B 24.955,C -1.5496,E1 25.006,E2 722.4095} C_DIS
LIN {X 8.2185,Y 138.2165,Z 161,A 82.4816,B 24.9552,C -1.5455,E1 25.011,E2 724.1821} C_DIS
LIN {X 12.8038,Y 137.8677,Z 161,A 80.4797,B 24.9556,C -1.54,E1 25.0166,E2 726.1959} C_DIS
LIN {X 16.9342,Y 137.4218,Z 161,A 78.8524,B 24.9553,C -1.5446,E1 25.0211,E2 727.811} C_DIS
LIN {X 21.1194,Y 136.8401,Z 161,A 77.247,B 24.9549,C -1.5519,E1 25.0254,E2 729.3978} C_DIS
LIN {X 27.3844,Y 135.7253,Z 161,A 74.8022,B 24.9543,C -1.5611,E1 25.0321,E2 731.8182} C_DIS
LIN {X 30.0036,Y 135.1726,Z 161,A 73.4786,B 24.9551,C -1.5487,E1 25.0358,E2 733.1694} C_DIS
LIN {X 32.9896,Y 134.4738,Z 161,A 72.2074,B 24.9551,C -1.5478,E1 25.0392,E2 734.4407} C_DIS
LIN {X 36.2647,Y 133.6279,Z 161,A 70.8079,B 24.9551,C -1.5469,E1 25.043,E2 735.8402} C_DIS
LIN {X 39.4455,Y 132.7236,Z 161,A 69.4357,B 24.9552,C -1.5457,E1 25.0467,E2 737.213} C_DIS
LIN {X 42.687,Y 131.7169,Z 161,A 68.032,B 24.9552,C -1.5446,E1 25.0504,E2 738.6167} C_DIS
LIN {X 46.5495,Y 130.4013,Z 161,A 66.2704,B 24.9556,C -1.5391,E1 25.0551,E2 740.3878} C_DIS
LIN {X 50.2085,Y 129.0359,Z 161,A 64.7496,B 24.9554,C -1.5427,E1 25.059,E2 741.8967} C_DIS
LIN {X 53.3054,Y 127.7876,Z 161,A 62.7804,B 24.9573,C -1.509,E1 25.0643,E2 743.941} C_DIS
LIN {X 57.774,Y 125.831,Z 161,A 61.5183,B 24.9551,C -1.5482,E1 25.0673,E2 745.1074} C_DIS
LIN {X 60.1608,Y 124.708,Z 161,A 60.2368,B 24.9558,C -1.5363,E1 25.0706,E2 746.4136} C_DIS
LIN {X 63.7064,Y 122.9357,Z 161,A 58.6182,B 24.9558,C -1.5353,E1 25.0746,E2 748.0302} C_DIS
LIN {X 67.3484,Y 120.9792,Z 161,A 56.781,B 24.9564,C -1.5259,E1 25.0791,E2 749.8844} C_DIS
LIN {X 70.9458,Y 118.9049,Z 161,A 55.0752,B 24.9564,C -1.524,E1 25.0833,E2 751.5895} C_DIS
LIN {X 74.7557,Y 116.5473,Z 161,A 53.2689,B 24.9565,C -1.5237,E1 25.0875,E2 753.3907} C_DIS
LIN {X 78.5521,Y 114.0232,Z 161,A 51.3491,B 24.9568,C -1.5186,E1 25.092,E2 755.3159} C_DIS
LIN {X 82.3688,Y 111.2979,Z 161,A 49.4131,B 24.957,C -1.5154,E1 25.0963,E2 757.2528} C_DIS
LIN {X 86.0778,Y 108.4542,Z 161,A 47.4903,B 24.9571,C -1.5124,E1 25.1006,E2 759.1755} C_DIS
LIN {X 89.7602,Y 105.4267,Z 161,A 45.6125,B 24.9571,C -1.5138,E1 25.1046,E2 761.0428} C_DIS
LIN {X 92.7537,Y 102.8036,Z 161,A 43.8827,B 24.9575,C -1.5058,E1 25.1082,E2 762.7847} C_DIS
LIN {X 96.2349,Y 99.5516,Z 161,A 42.0143,B 24.9575,C -1.5073,E1 25.112,E2 764.6417} C_DIS
LIN {X 99.1952,Y 96.603,Z 161,A 40.1876,B 24.958,C -1.498,E1 25.1156,E2 766.4827} C_DIS
LIN {X 102.4848,Y 93.105,Z 161,A 38.2743,B 24.958,C -1.4976,E1 25.1192,E2 768.3885} C_DIS
LIN {X 105.4998,Y 89.6742,Z 161,A 36.4538,B 24.958,C -1.497,E1 25.1225,E2 770.2022} C_DIS
LIN {X 108.1633,Y 86.4433,Z 161,A 34.6379,B 24.9585,C -1.488,E1 25.1257,E2 772.0307} C_DIS
LIN {X 110.9608,Y 82.8215,Z 161,A 32.7545,B 24.9588,C -1.4839,E1 25.1289,E2 773.9151} C_DIS
LIN {X 113.6919,Y 79.0306,Z 161,A 30.8437,B 24.959,C -1.4801,E1 25.132,E2 775.8253} C_DIS
LIN {X 116.1403,Y 75.3863,Z 161,A 29.0129,B 24.9593,C -1.4745,E1 25.1348,E2 777.6603} C_DIS
LIN {X 118.6755,Y 71.3297,Z 161,A 27.1507,B 24.9592,C -1.4758,E1 25.1375,E2 779.51} C_DIS
LIN {X 120.7827,Y 67.6996,Z 161,A 25.3102,B 24.9598,C -1.465,E1 25.1401,E2 781.3663} C_DIS
LIN {X 123.0645,Y 63.4568,Z 161,A 23.4658,B 24.9596,C -1.4679,E1 25.1425,E2 783.1942} C_DIS
LIN {X 124.5451,Y 60.5007,Z 161,A 22.09,B 24.9599,C -1.4635,E1 25.1442,E2 784.5731} C_DIS
LIN {X 125.9385,Y 57.5415,Z 161,A 20.7427,B 24.9601,C -1.4599,E1 25.1458,E2 785.9216} C_DIS
LIN {X 127.1196,Y 54.8794,Z 161,A 19.4975,B 24.9604,C -1.4541,E1 25.1472,E2 787.1737} C_DIS
LIN {X 128.5337,Y 51.4813,Z 161,A 18.0028,B 24.9606,C -1.4511,E1 25.1488,E2 788.6671} C_DIS
LIN {X 129.9229,Y 47.8722,Z 161,A 16.4593,B 24.9606,C -1.4495,E1 25.1503,E2 790.2058} C_DIS
LIN {X 130.9739,Y 44.9136,Z 161,A 15.1625,B 24.9608,C -1.4457,E1 25.1515,E2 791.5043} C_DIS
LIN {X 131.9705,Y 41.893,Z 161,A 13.8169,B 24.9612,C -1.4399,E1 25.1526,E2 792.8559} C_DIS
LIN {X 133.0343,Y 38.3843,Z 161,A 12.3466,B 24.9612,C -1.4378,E1 25.1538,E2 794.3227} C_DIS
LIN {X 133.9313,Y 35.1271,Z 161,A 10.958,B 24.9615,C -1.434,E1 25.1548,E2 795.7124} C_DIS
LIN {X 134.6661,Y 32.1917,Z 161,A 9.6786,B 24.9618,C -1.4284,E1 25.1557,E2 796.9975} C_DIS
LIN {X 135.3734,Y 29.0734,Z 161,A 8.3652,B 24.962,C -1.4247,E1 25.1565,E2 798.3119} C_DIS
LIN {X 136.0824,Y 25.5539,Z 161,A 6.918,B 24.9621,C -1.4222,E1 25.1572,E2 799.7567} C_DIS
LIN {X 136.6803,Y 22.1396,Z 161,A 5.5038,B 24.9623,C -1.4187,E1 25.1579,E2 801.1709} C_DIS
LIN {X 137.2893,Y 17.9686,Z 161,A 3.7479,B 24.9626,C -1.4123,E1 25.1586,E2 802.9314} C_DIS
LIN {X 137.7138,Y 14.3654,Z 161,A 2.1512,B 24.9632,C -1.4019,E1 25.1591,E2 804.5432} C_DIS
LIN {X 138.245,Y 7.7527,Z 161,A -0.5525,B 24.9635,C -1.3952,E1 25.1596,E2 807.2467} C_DIS
LIN {X 138.4083,Y 3.7995,Z 161,A -2.1106,B 24.9635,C -1.3943,E1 25.1598,E2 808.7975} C_DIS
LIN {X 138.4619,Y -0.1987,Z 161,A -3.8458,B 24.9641,C -1.3841,E1 25.1598,E2 810.5463} C_DIS
LIN {X 138.4053,Y -3.9056,Z 161,A -5.267,B 24.9641,C -1.3856,E1 25.1597,E2 811.9557} C_DIS
LIN {X 138.2441,Y -7.7707,Z 161,A -6.801,B 24.9641,C -1.3841,E1 25.1595,E2 813.4841} C_DIS
LIN {X 137.9385,Y -12.0152,Z 161,A -8.5953,B 24.9645,C -1.3763,E1 25.1591,E2 815.2861} C_DIS
LIN {X 137.6123,Y -15.3088,Z 161,A -9.9303,B 24.9647,C -1.3738,E1 25.1587,E2 816.6193} C_DIS
LIN {X 137.2196,Y -18.5008,Z 161,A -11.5795,B 24.9658,C -1.3509,E1 25.1581,E2 818.3125} C_DIS
LIN {X 136.7104,Y -21.9565,Z 161,A -12.6847,B 24.9651,C -1.3658,E1 25.1576,E2 819.3763} C_DIS
LIN {X 136.1811,Y -25.027,Z 161,A -13.9783,B 24.9653,C -1.3612,E1 25.157,E2 820.6728} C_DIS
LIN {X 135.5243,Y -28.3722,Z 161,A -15.3784,B 24.9655,C -1.3572,E1 25.1562,E2 822.0744} C_DIS
LIN {X 134.7326,Y -31.9156,Z 161,A -16.9788,B 24.966,C -1.3466,E1 25.1552,E2 823.6904} C_DIS
LIN {X 133.7627,Y -35.7592,Z 161,A -18.5104,B 24.966,C -1.3475,E1 25.1541,E2 825.2111} C_DIS
LIN {X 132.7778,Y -39.2601,Z 161,A -20.0842,B 24.9664,C -1.3386,E1 25.1529,E2 826.7969} C_DIS
LIN {X 131.6152,Y -43.0026,Z 161,A -21.5898,B 24.9664,C -1.3401,E1 25.1517,E2 828.2905} C_DIS
LIN {X 130.6695,Y -45.7915,Z 161,A -22.8306,B 24.9666,C -1.3349,E1 25.1505,E2 829.5365} C_DIS
LIN {X 129.2479,Y -49.663,Z 161,A -24.6601,B 24.9673,C -1.3223,E1 25.1487,E2 831.3853} C_DIS
LIN {X 127.7184,Y -53.4711,Z 161,A -26.2815,B 24.9673,C -1.3214,E1 25.147,E2 833} C_DIS
LIN {X 125.9313,Y -57.5571,Z 161,A -27.9542,B 24.9671,C -1.3256,E1 25.1451,E2 834.6538} C_DIS
LIN {X 123.9712,Y -61.6641,Z 161,A -30.0463,B 24.968,C -1.3077,E1 25.1425,E2 836.7768} C_DIS
LIN {X 121.7406,Y -65.9626,Z 161,A -32.0285,B 24.9682,C -1.3028,E1 25.1399,E2 838.7601} C_DIS
LIN {X 119.4472,Y -70.029,Z 161,A -33.9413,B 24.9684,C -1.2981,E1 25.1373,E2 840.674} C_DIS
LIN {X 116.9784,Y -74.0794,Z 161,A -35.9,B 24.9687,C -1.2926,E1 25.1344,E2 842.6359} C_DIS
LIN {X 114.3431,Y -78.0861,Z 161,A -37.7484,B 24.9687,C -1.2947,E1 25.1315,E2 844.4701} C_DIS
LIN {X 112.0873,Y -81.2903,Z 161,A -39.4894,B 24.9692,C -1.2832,E1 25.1287,E2 846.2297} C_DIS
LIN {X 109.1345,Y -85.2144,Z 161,A -41.405,B 24.9692,C -1.2843,E1 25.1255,E2 848.1338} C_DIS
LIN {X 106.4712,Y -88.5191,Z 161,A -43.1302,B 24.9692,C -1.2813,E1 25.1224,E2 849.858} C_DIS
LIN {X 103.8216,Y -91.612,Z 161,A -44.8065,B 24.9694,C -1.2773,E1 25.1193,E2 851.5361} C_DIS
LIN {X 101.4902,Y -94.1884,Z 161,A -46.3582,B 24.9699,C -1.267,E1 25.1164,E2 853.1052} C_DIS
LIN {X 98.5141,Y -97.2975,Z 161,A -48.1213,B 24.9701,C -1.2635,E1 25.1129,E2 854.8691} C_DIS
LIN {X 95.1355,Y -100.6028,Z 161,A -49.9778,B 24.9701,C -1.2643,E1 25.1092,E2 856.7157} C_DIS
LIN {X 91.9793,Y -103.4969,Z 161,A -51.7407,B 24.9702,C -1.2606,E1 25.1056,E2 858.4804} C_DIS
LIN {X 88.7964,Y -106.24,Z 161,A -53.4623,B 24.9704,C -1.2575,E1 25.1019,E2 860.2026} C_DIS
LIN {X 85.5663,Y -108.8581,Z 161,A -55.2815,B 24.9708,C -1.248,E1 25.0979,E2 862.0374} C_DIS
LIN {X 82.241,Y -111.3921,Z 161,A -57.0077,B 24.971,C -1.2445,E1 25.0941,E2 863.7658} C_DIS
LIN {X 78.8811,Y -113.7959,Z 161,A -58.5951,B 24.9708,C -1.2478,E1 25.0905,E2 865.3398} C_DIS
LIN {X 75.4272,Y -116.1138,Z 161,A -60.33,B 24.971,C -1.2435,E1 25.0864,E2 867.079} C_DIS
LIN {X 71.8415,Y -118.3661,Z 161,A -62.1544,B 24.9714,C -1.236,E1 25.082,E2 868.9154} C_DIS
LIN {X 67.7253,Y -120.7683,Z 161,A -64.1295,B 24.9716,C -1.2322,E1 25.0773,E2 870.8936} C_DIS
LIN {X 63.4892,Y -123.048,Z 161,A -65.9676,B 24.9713,C -1.2373,E1 25.0728,E2 872.7144} C_DIS
LIN {X 60.9492,Y -124.3239,Z 161,A -67.199,B 24.9716,C -1.2323,E1 25.0697,E2 873.9545} C_DIS
LIN {X 57.9246,Y -125.7613,Z 161,A -68.5715,B 24.9716,C -1.2308,E1 25.0662,E2 875.3269} C_DIS
LIN {X 54.2184,Y -127.4054,Z 161,A -70.2112,B 24.9716,C -1.2303,E1 25.062,E2 876.9639} C_DIS
LIN {X 50.9485,Y -128.7482,Z 161,A -71.6651,B 24.9717,C -1.2286,E1 25.0582,E2 878.4184} C_DIS
LIN {X 48.204,Y -129.7986,Z 161,A -72.9056,B 24.9719,C -1.2256,E1 25.055,E2 879.6634} C_DIS
LIN {X 44.8582,Y -130.993,Z 161,A -74.3394,B 24.9719,C -1.2256,E1 25.0512,E2 881.094} C_DIS
LIN {X 41.7708,Y -132.0095,Z 161,A -75.6851,B 24.9719,C -1.224,E1 25.0476,E2 882.4413} C_DIS
LIN {X 37.8963,Y -133.1745,Z 161,A -77.3369,B 24.9719,C -1.2233,E1 25.0432,E2 884.0919} C_DIS
LIN {X 34.8737,Y -133.9988,Z 161,A -78.7516,B 24.9723,C -1.2153,E1 25.0393,E2 885.5233} C_DIS
LIN {X 31.1041,Y -134.9215,Z 161,A -80.3688,B 24.9724,C -1.2131,E1 25.0349,E2 887.1434} C_DIS
LIN {X 27.1624,Y -135.7705,Z 161,A -81.9189,B 24.9722,C -1.2181,E1 25.0307,E2 888.6796} C_DIS
LIN {X 23.2571,Y -136.4938,Z 161,A -83.4255,B 24.9719,C -1.2244,E1 25.0266,E2 890.1698} C_DIS
LIN {X 20.073,Y -136.9984,Z 161,A -84.9736,B 24.9725,C -1.2115,E1 25.0223,E2 891.7468} C_DIS
LIN {X 14.6211,Y -137.6863,Z 161,A -87.0964,B 24.9722,C -1.2185,E1 25.0165,E2 893.8516} C_DIS
LIN {X 11.3059,Y -137.9984,Z 161,A -88.6446,B 24.9727,C -1.2083,E1 25.0121,E2 895.4229} C_DIS
LIN {X 6.9272,Y -138.287,Z 161,A -90.3244,B 24.9724,C -1.2151,E1 25.0074,E2 897.0861} C_DIS
LIN {X 3.2791,Y -138.4227,Z 161,A -91.9855,B 24.9728,C -1.2063,E1 25.0028,E2 898.7676} C_DIS
LIN {X 3.2791,Y -138.4227,Z 161,A -91.9855,B 24.9728,C -1.2063,E1 25.0028,E2 898.7676} C_DIS
Enddeposition()
LIN {X 0.972,Y -137.5286,Z 161,A -92.7717,B 24.9716,C -1.2317,E1 25.0007,E2 899.4936} C_DIS
Startdeposition()
$VEL.CP = VEL_PRINT
LIN {X 3.8326,Y -137.4828,Z 161,A -91.0238,B 24.9702,C -1.2625,E1 25.0058,E2 897.6731} C_DIS
LIN {X 7.9453,Y -137.3074,Z 161,A -88.4471,B 24.9678,C -1.3112,E1 25.0133,E2 894.9819} C_DIS
LIN {X 14.3573,Y -136.7851,Z 161,A -86.7232,B 24.9703,C -1.2592,E1 25.0178,E2 893.3821} C_DIS
LIN {X 20.7196,Y -135.9668,Z 161,A -84.168,B 24.9705,C -1.2545,E1 25.0248,E2 890.8403} C_DIS
LIN {X 25.9543,Y -135.0649,Z 161,A -81.7749,B 24.97,C -1.2663,E1 25.0314,E2 888.4218} C_DIS
LIN {X 29.3967,Y -134.3581,Z 161,A -80.3343,B 24.97,C -1.2663,E1 25.0354,E2 886.9831} C_DIS
LIN {X 32.7102,Y -133.5904,Z 161,A -78.784,B 24.9695,C -1.2752,E1 25.0396,E2 885.4139} C_DIS
LIN {X 37.6041,Y -132.2965,Z 161,A -76.8165,B 24.9698,C -1.2696,E1 25.0449,E2 883.4629} C_DIS
LIN {X 40.6751,Y -131.3843,Z 161,A -75.4487,B 24.9696,C -1.273,E1 25.0486,E2 882.0893} C_DIS
LIN {X 44.105,Y -130.274,Z 161,A -73.9574,B 24.9696,C -1.2743,E1 25.0525,E2 880.5978} C_DIS
LIN {X 50.3527,Y -127.9882,Z 161,A -71.0704,B 24.9691,C -1.2847,E1 25.0601,E2 877.6925} C_DIS
LIN {X 55.7918,Y -125.712,Z 161,A -68.9117,B 24.9697,C -1.2716,E1 25.0656,E2 875.5699} C_DIS
LIN {X 59.2768,Y -124.1061,Z 161,A -66.8644,B 24.9684,C -1.2996,E1 25.0709,E2 873.4616} C_DIS
LIN {X 62.2211,Y -122.6565,Z 161,A -66.0302,B 24.9697,C -1.2717,E1 25.0728,E2 872.6957} C_DIS
LIN {X 65.9369,Y -120.7018,Z 161,A -63.9505,B 24.9687,C -1.2935,E1 25.078,E2 870.5703} C_DIS
LIN {X 69.8195,Y -118.4984,Z 161,A -62.1021,B 24.9685,C -1.2963,E1 25.0825,E2 868.7209} C_DIS
LIN {X 73.3006,Y -116.3771,Z 161,A -60.4755,B 24.9685,C -1.2955,E1 25.0864,E2 867.1013} C_DIS
LIN {X 76.6981,Y -114.1672,Z 161,A -58.7334,B 24.9682,C -1.302,E1 25.0904,E2 865.3497} C_DIS
LIN {X 80.2142,Y -111.7245,Z 161,A -56.9744,B 24.9682,C -1.3044,E1 25.0944,E2 863.5912} C_DIS
LIN {X 83.5919,Y -109.2199,Z 161,A -55.2334,B 24.968,C -1.3076,E1 25.0983,E2 861.8489} C_DIS
LIN {X 86.8564,Y -106.6425,Z 161,A -53.4728,B 24.9677,C -1.3131,E1 25.1022,E2 860.0818} C_DIS
LIN {X 90.2444,Y -103.7911,Z 161,A -51.6483,B 24.9675,C -1.3163,E1 25.106,E2 858.2571} C_DIS
LIN {X 93.5393,Y -100.8319,Z 161,A -49.8051,B 24.9673,C -1.3206,E1 25.1099,E2 856.411} C_DIS
LIN {X 96.7137,Y -97.7914,Z 161,A -47.9543,B 24.9671,C -1.3263,E1 25.1136,E2 854.5546} C_DIS
LIN {X 99.8058,Y -94.6336,Z 161,A -46.163,B 24.967,C -1.3281,E1 25.117,E2 852.7666} C_DIS
LIN {X 102.8064,Y -91.365,Z 161,A -44.325,B 24.9667,C -1.3324,E1 25.1205,E2 850.9268} C_DIS
LIN {X 105.6651,Y -88.0435,Z 161,A -42.4926,B 24.9665,C -1.3377,E1 25.1238,E2 849.0903} C_DIS
LIN {X 108.446,Y -84.5946,Z 161,A -40.6261,B 24.9662,C -1.344,E1 25.127,E2 847.2177} C_DIS
LIN {X 111.135,Y -81.0293,Z 161,A -38.7994,B 24.966,C -1.3472,E1 25.1301,E2 845.392} C_DIS
LIN {X 114.3013,Y -76.4972,Z 161,A -36.4499,B 24.9655,C -1.3565,E1 25.1338,E2 843.0322} C_DIS
LIN {X 116.9153,Y -72.4395,Z 161,A -34.5755,B 24.9656,C -1.3545,E1 25.1366,E2 841.1721} C_DIS
LIN {X 119.024,Y -68.9195,Z 161,A -32.8393,B 24.9653,C -1.3612,E1 25.139,E2 839.429} C_DIS
LIN {X 121.1544,Y -65.1016,Z 161,A -30.9069,B 24.9647,C -1.3732,E1 25.1416,E2 837.4786} C_DIS
LIN {X 122.8628,Y -61.816,Z 161,A -29.6066,B 24.9652,C -1.3638,E1 25.1433,E2 836.2072} C_DIS
LIN {X 124.1551,Y -59.1742,Z 161,A -28.3164,B 24.9648,C -1.3714,E1 25.1448,E2 834.906} C_DIS
LIN {X 126.8243,Y -53.2138,Z 161,A -25.8579,B 24.9651,C -1.3646,E1 25.1476,E2 832.4768} C_DIS
LIN {X 127.9121,Y -50.5482,Z 161,A -24.246,B 24.9637,C -1.3924,E1 25.1493,E2 830.8084} C_DIS
LIN {X 129.6203,Y -45.9907,Z 161,A -22.388,B 24.9639,C -1.389,E1 25.151,E2 828.9688} C_DIS
LIN {X 130.9452,Y -42.0654,Z 161,A -20.6307,B 24.9635,C -1.3965,E1 25.1526,E2 827.204} C_DIS
LIN {X 132.1,Y -38.2862,Z 161,A -19.1292,B 24.9636,C -1.3934,E1 25.1538,E2 825.7183} C_DIS
LIN {X 133.1236,Y -34.566,Z 161,A -17.3852,B 24.9629,C -1.4066,E1 25.155,E2 823.9532} C_DIS
LIN {X 134.0599,Y -30.7258,Z 161,A -15.8657,B 24.963,C -1.4046,E1 25.156,E2 822.4472} C_DIS
LIN {X 134.791,Y -27.3409,Z 161,A -14.4374,B 24.9628,C -1.4085,E1 25.1568,E2 821.0179} C_DIS
LIN {X 135.4539,Y -23.8439,Z 161,A -12.9416,B 24.9625,C -1.4142,E1 25.1576,E2 819.5175} C_DIS
LIN {X 136.3565,Y -17.9742,Z 161,A -10.2832,B 24.9615,C -1.4332,E1 25.1586,E2 816.8301} C_DIS
LIN {X 137.0029,Y -12.1111,Z 161,A -7.9832,B 24.9615,C -1.4321,E1 25.1593,E2 814.5461} C_DIS
LIN {X 137.2713,Y -8.531,Z 161,A -6.5154,B 24.9614,C -1.4355,E1 25.1596,E2 813.0791} C_DIS
LIN {X 137.5196,Y -2.1424,Z 161,A -3.663,B 24.9603,C -1.4554,E1 25.1598,E2 810.1968} C_DIS
LIN {X 137.5322,Y 1.1719,Z 161,A -2.2998,B 24.9601,C -1.459,E1 25.1598,E2 808.8333} C_DIS
LIN {X 137.4675,Y 4.382,Z 161,A -0.4087,B 24.9581,C -1.4959,E1 25.1596,E2 806.8663} C_DIS
LIN {X 137.1239,Y 10.6609,Z 161,A 1.2533,B 24.9607,C -1.4485,E1 25.1593,E2 805.326} C_DIS
LIN {X 136.6782,Y 15.3513,Z 161,A 3.245,B 24.9603,C -1.4566,E1 25.1587,E2 803.3271} C_DIS
LIN {X 136.0561,Y 20.1333,Z 161,A 5.2476,B 24.9599,C -1.4628,E1 25.1579,E2 801.3217} C_DIS
LIN {X 135.3633,Y 24.3502,Z 161,A 7.0879,B 24.9594,C -1.4721,E1 25.1571,E2 799.4703} C_DIS
LIN {X 134.7247,Y 27.6668,Z 161,A 8.4471,B 24.9594,C -1.4738,E1 25.1563,E2 798.1149} C_DIS
LIN {X 134.0583,Y 30.7326,Z 161,A 9.7688,B 24.959,C -1.4788,E1 25.1555,E2 796.789} C_DIS
LIN {X 133.2643,Y 34.0114,Z 161,A 11.1555,B 24.9588,C -1.4822,E1 25.1546,E2 795.4023} C_DIS
LIN {X 132.3453,Y 37.4299,Z 161,A 12.621,B 24.9586,C -1.4863,E1 25.1535,E2 793.9356} C_DIS
LIN {X 130.4873,Y 43.4645,Z 161,A 14.9243,B 24.9592,C -1.4756,E1 25.1517,E2 791.6706} C_DIS
LIN {X 129.3015,Y 46.8751,Z 161,A 16.76,B 24.9579,C -1.4993,E1 25.1499,E2 789.7894} C_DIS
LIN {X 128.1115,Y 50.0357,Z 161,A 18.1114,B 24.9579,C -1.5004,E1 25.1485,E2 788.443} C_DIS
LIN {X 126.7357,Y 53.4259,Z 161,A 19.6305,B 24.9576,C -1.5046,E1 25.1469,E2 786.9223} C_DIS
LIN {X 125.3734,Y 56.5487,Z 161,A 21.0654,B 24.9573,C -1.5097,E1 25.1453,E2 785.4832} C_DIS
LIN {X 123.9591,Y 59.5843,Z 161,A 22.4191,B 24.9573,C -1.5114,E1 25.1437,E2 784.1328} C_DIS
LIN {X 122.4431,Y 62.6404,Z 161,A 23.8521,B 24.9569,C -1.5162,E1 25.1419,E2 782.6961} C_DIS
LIN {X 120.8101,Y 65.7383,Z 161,A 25.383,B 24.9565,C -1.5244,E1 25.1398,E2 781.1539} C_DIS
LIN {X 118.6477,Y 69.5653,Z 161,A 27.1997,B 24.9562,C -1.5287,E1 25.1373,E2 779.3365} C_DIS
LIN {X 116.3865,Y 73.2858,Z 161,A 29.0418,B 24.9558,C -1.5352,E1 25.1346,E2 777.4883} C_DIS
LIN {X 113.9033,Y 77.0884,Z 161,A 31.1118,B 24.955,C -1.5505,E1 25.1313,E2 775.3927} C_DIS
LIN {X 111.9987,Y 79.8306,Z 161,A 32.1296,B 24.956,C -1.5327,E1 25.1298,E2 774.4217} C_DIS
LIN {X 109.9816,Y 82.5878,Z 161,A 33.6515,B 24.9555,C -1.542,E1 25.1272,E2 772.8853} C_DIS
LIN {X 107.3693,Y 85.9569,Z 161,A 35.2685,B 24.9557,C -1.5373,E1 25.1244,E2 771.2869} C_DIS
LIN {X 105.1867,Y 88.6139,Z 161,A 36.8936,B 24.9549,C -1.5518,E1 25.1215,E2 769.6352} C_DIS
LIN {X 102.1632,Y 92.084,Z 161,A 38.6427,B 24.9552,C -1.5467,E1 25.1183,E2 767.9058} C_DIS
LIN {X 99.8033,Y 94.6362,Z 161,A 40.2285,B 24.9545,C -1.5578,E1 25.1152,E2 766.3006} C_DIS
LIN {X 96.8322,Y 97.6737,Z 161,A 42.072,B 24.9541,C -1.5659,E1 25.1116,E2 764.4459} C_DIS
LIN {X 93.3282,Y 101.0275,Z 161,A 43.9914,B 24.9541,C -1.5645,E1 25.1077,E2 762.5378} C_DIS
LIN {X 90.0975,Y 103.9193,Z 161,A 46.1955,B 24.9526,C -1.5907,E1 25.103,E2 760.2804} C_DIS
LIN {X 86.8638,Y 106.6364,Z 161,A 47.5623,B 24.9537,C -1.5719,E1 25.1001,E2 758.9632} C_DIS
LIN {X 83.5738,Y 109.2338,Z 161,A 49.2879,B 24.9536,C -1.574,E1 25.0963,E2 757.239} C_DIS
LIN {X 80.0377,Y 111.8506,Z 161,A 51.1062,B 24.9534,C -1.5765,E1 25.0922,E2 755.4212} C_DIS
LIN {X 76.604,Y 114.2301,Z 161,A 52.8278,B 24.9534,C -1.5784,E1 25.0882,E2 753.701} C_DIS
LIN {X 73.0241,Y 116.5515,Z 161,A 54.6331,B 24.9531,C -1.5829,E1 25.084,E2 751.891} C_DIS
LIN {X 69.3279,Y 118.7872,Z 161,A 56.465,B 24.9528,C -1.5874,E1 25.0796,E2 750.0541} C_DIS
LIN {X 65.4249,Y 120.9807,Z 161,A 58.3321,B 24.9526,C -1.5902,E1 25.075,E2 748.1858} C_DIS
LIN {X 62.1613,Y 122.6869,Z 161,A 59.7466,B 24.9529,C -1.5856,E1 25.0715,E2 746.786} C_DIS
LIN {X 58.9556,Y 124.2595,Z 161,A 61.2351,B 24.9528,C -1.5875,E1 25.0678,E2 745.2969} C_DIS
LIN {X 54.9707,Y 126.0733,Z 161,A 63.0916,B 24.9525,C -1.5915,E1 25.063,E2 743.4356} C_DIS
LIN {X 50.8548,Y 127.7898,Z 161,A 64.8789,B 24.9527,C -1.5896,E1 25.0584,E2 741.6569} C_DIS
LIN {X 47.7397,Y 128.9856,Z 161,A 66.3753,B 24.9522,C -1.5968,E1 25.0545,E2 740.1467} C_DIS
LIN {X 43.4023,Y 130.508,Z 161,A 68.231,B 24.9523,C -1.5952,E1 25.0496,E2 738.2983} C_DIS
LIN {X 39.9636,Y 131.602,Z 161,A 69.6998,B 24.9523,C -1.5945,E1 25.0457,E2 736.8337} C_DIS
LIN {X 36.1652,Y 132.698,Z 161,A 71.4575,B 24.9519,C -1.6018,E1 25.0409,E2 735.062} C_DIS
LIN {X 32.3663,Y 133.6733,Z 161,A 73.0019,B 24.9522,C -1.5979,E1 25.0368,E2 733.5289} C_DIS
LIN {X 28.6467,Y 134.52,Z 161,A 74.5578,B 24.9522,C -1.5969,E1 25.0325,E2 731.9775} C_DIS
LIN {X 23.6587,Y 135.4871,Z 161,A 77.0555,B 24.9509,C -1.6186,E1 25.0255,E2 729.4312} C_DIS
LIN {X 19.9259,Y 136.0858,Z 161,A 78.4788,B 24.9514,C -1.6107,E1 25.0217,E2 728.0277} C_DIS
LIN {X 14.9278,Y 136.7237,Z 161,A 81.0625,B 24.9497,C -1.6376,E1 25.0143,E2 725.3821} C_DIS
LIN {X 9.2327,Y 137.228,Z 161,A 82.9885,B 24.9513,C -1.6128,E1 25.0091,E2 723.5159} C_DIS
LIN {X 2.5737,Y 137.5124,Z 161,A 86.3858,B 24.9492,C -1.6463,E1 24.9994,E2 720.0398} C_DIS
LIN {X -3.9241,Y 137.4802,Z 161,A 88.8133,B 24.9502,C -1.6303,E1 24.9927,E2 717.65} C_DIS
LIN {X -8.9463,Y 137.2458,Z 161,A 90.1084,B 24.9528,C -1.5864,E1 24.9894,E2 716.4585} C_DIS
LIN {X -16.9247,Y 136.4922,Z 161,A 93.5834,B 24.9525,C -1.5919,E1 24.9797,E2 712.9686} C_DIS
LIN {X -21.2909,Y 135.8783,Z 161,A 95.5074,B 24.9523,C -1.5953,E1 24.9744,E2 711.035} C_DIS
LIN {X -25.4704,Y 135.1574,Z 161,A 97.3322,B 24.9523,C -1.597,E1 24.9694,E2 709.2042} C_DIS
LIN {X -29.1448,Y 134.4125,Z 161,A 98.8195,B 24.9525,C -1.5917,E1 24.9653,E2 707.7278} C_DIS
LIN {X -32.4366,Y 133.6564,Z 161,A 100.2473,B 24.9525,C -1.5914,E1 24.9614,E2 706.2987} C_DIS
LIN {X -36.3103,Y 132.6584,Z 161,A 102.3186,B 24.9514,C -1.6112,E1 24.9557,E2 704.1775} C_DIS
LIN {X -39.9889,Y 131.5943,Z 161,A 103.5971,B 24.9525,C -1.5925,E1 24.9524,E2 702.9409} C_DIS
LIN {X -43.891,Y 130.3453,Z 161,A 105.1887,B 24.953,C -1.5844,E1 24.9482,E2 701.3659} C_DIS
LIN {X -47.0102,Y 129.2527,Z 161,A 106.6755,B 24.9527,C -1.5884,E1 24.9443,E2 699.8666} C_DIS
LIN {X -53.1107,Y 126.8674,Z 161,A 109.3361,B 24.9532,C -1.5809,E1 24.9374,E2 697.2178} C_DIS
LIN {X -56.3628,Y 125.4565,Z 161,A 110.842,B 24.9532,C -1.5802,E1 24.9336,E2 695.71} C_DIS
LIN {X -59.5788,Y 123.9618,Z 161,A 112.3543,B 24.9532,C -1.5797,E1 24.9297,E2 694.1952} C_DIS
LIN {X -63.2339,Y 122.1399,Z 161,A 115.2704,B 24.9495,C -1.6409,E1 24.9222,E2 691.1255} C_DIS
LIN {X -70.7165,Y 117.9656,Z 161,A 117.6847,B 24.9536,C -1.5733,E1 24.9167,E2 688.8647} C_DIS
LIN {X -74.7867,Y 115.4278,Z 161,A 119.4887,B 24.9544,C -1.5593,E1 24.9125,E2 687.0882} C_DIS
LIN {X -77.0639,Y 113.9199,Z 161,A 120.8043,B 24.954,C -1.5662,E1 24.9094,E2 685.7517} C_DIS
LIN {X -80.6862,Y 111.3837,Z 161,A 122.6723,B 24.9542,C -1.5637,E1 24.9052,E2 683.8832} C_DIS
LIN {X -84.2693,Y 108.6981,Z 161,A 124.5903,B 24.9542,C -1.5624,E1 24.9009,E2 681.9614} C_DIS
LIN {X -86.9934,Y 106.5305,Z 161,A 125.996,B 24.9546,C -1.5569,E1 24.8979,E2 680.5636} C_DIS
LIN {X -90.4109,Y 103.6458,Z 161,A 127.8759,B 24.9548,C -1.5534,E1 24.8939,E2 678.6847} C_DIS
LIN {X -93.5472,Y 100.8245,Z 161,A 129.6506,B 24.955,C -1.5501,E1 24.8902,E2 676.9106} C_DIS
LIN {X -96.6673,Y 97.8374,Z 161,A 131.4455,B 24.9553,C -1.5455,E1 24.8866,E2 675.1194} C_DIS
LIN {X -99.6886,Y 94.7572,Z 161,A 133.2904,B 24.9553,C -1.5434,E1 24.8831,E2 673.2715} C_DIS
LIN {X -102.7016,Y 91.4829,Z 161,A 135.1481,B 24.9556,C -1.5388,E1 24.8796,E2 671.4165} C_DIS
LIN {X -106.4961,Y 87.0354,Z 161,A 137.6955,B 24.9556,C -1.538,E1 24.875,E2 668.8591} C_DIS
LIN {X -109.6004,Y 83.093,Z 161,A 139.6344,B 24.9565,C -1.5245,E1 24.8717,E2 666.9432} C_DIS
LIN {X -111.8682,Y 80.0131,Z 161,A 141.2644,B 24.9566,C -1.5219,E1 24.8691,E2 665.3115} C_DIS
LIN {X -114.3444,Y 76.4327,Z 161,A 143.0995,B 24.9568,C -1.5178,E1 24.8662,E2 663.477} C_DIS
LIN {X -117.201,Y 71.9759,Z 161,A 145.2906,B 24.9572,C -1.5107,E1 24.8629,E2 661.2917} C_DIS
LIN {X -119.3276,Y 68.393,Z 161,A 147.2566,B 24.9569,C -1.5173,E1 24.8601,E2 659.2998} C_DIS
LIN {X -120.893,Y 65.5864,Z 161,A 148.1344,B 24.9584,C -1.4897,E1 24.8591,E2 658.4829} C_DIS
LIN {X -122.8076,Y 61.9243,Z 161,A 150.1547,B 24.9579,C -1.4997,E1 24.8564,E2 656.4281} C_DIS
LIN {X -124.3194,Y 58.8302,Z 161,A 151.5036,B 24.9584,C -1.4909,E1 24.8548,E2 655.0928} C_DIS
LIN {X -125.6874,Y 55.8467,Z 161,A 152.8822,B 24.9586,C -1.4873,E1 24.8532,E2 653.7153} C_DIS
LIN {X -127.0386,Y 52.7007,Z 161,A 154.3172,B 24.9588,C -1.4832,E1 24.8517,E2 652.2821} C_DIS
LIN {X -128.2872,Y 49.5836,Z 161,A 155.7114,B 24.959,C -1.4786,E1 24.8502,E2 650.8911} C_DIS
LIN {X -129.4507,Y 46.461,Z 161,A 157.1324,B 24.9592,C -1.4758,E1 24.8489,E2 649.4687} C_DIS
LIN {X -130.6853,Y 42.8699,Z 161,A 158.8274,B 24.9592,C -1.4765,E1 24.8474,E2 647.7625} C_DIS
LIN {X -132.0051,Y 38.6102,Z 161,A 160.6083,B 24.9597,C -1.4666,E1 24.8459,E2 645.9948} C_DIS
LIN {X -133.0011,Y 35.029,Z 161,A 162.2795,B 24.9597,C -1.4677,E1 24.8447,E2 644.3111} C_DIS
LIN {X -134.0257,Y 30.8755,Z 161,A 163.9714,B 24.9602,C -1.4573,E1 24.8436,E2 642.6342} C_DIS
LIN {X -134.8534,Y 27.0343,Z 161,A 165.5334,B 24.9607,C -1.4481,E1 24.8428,E2 641.0848} C_DIS
LIN {X -135.412,Y 24.0779,Z 161,A 166.9314,B 24.9605,C -1.4513,E1 24.842,E2 639.6708} C_DIS
LIN {X -136.1152,Y 19.72,Z 161,A 168.7205,B 24.961,C -1.4427,E1 24.8413,E2 637.8917} C_DIS
LIN {X -136.6092,Y 15.9443,Z 161,A 170.3629,B 24.9611,C -1.4403,E1 24.8407,E2 636.2452} C_DIS
LIN {X -137.0416,Y 11.6531,Z 161,A 172.1098,B 24.9616,C -1.4318,E1 24.8403,E2 634.5081} C_DIS
LIN {X -137.2997,Y 8.0713,Z 161,A 173.6096,B 24.9619,C -1.427,E1 24.84,E2 633.0107} C_DIS
LIN {X -137.4791,Y 3.9638,Z 161,A 175.3965,B 24.9619,C -1.4251,E1 24.8398,E2 631.2176} C_DIS
LIN {X -137.538,Y -0.1217,Z 161,A 177.1536,B 24.9621,C -1.4222,E1 24.8398,E2 629.4568} C_DIS
LIN {X -137.4761,Y -4.074,Z 161,A 178.7909,B 24.9624,C -1.4163,E1 24.8399,E2 627.8237} C_DIS
LIN {X -137.2761,Y -8.4531,Z 161,A -179.4671,B 24.963,C -1.406,E1 24.8402,E2 626.0958} C_DIS
LIN {X -137.0213,Y -11.8929,Z 161,A -178.0284,B 24.9632,C -1.4013,E1 24.8405,E2 624.6596} C_DIS
LIN {X -136.6731,Y -15.3983,Z 161,A -176.4076,B 24.9631,C -1.4043,E1 24.841,E2 623.0219} C_DIS
LIN {X -136.1628,Y -19.387,Z 161,A -174.8342,B 24.9636,C -1.3937,E1 24.8415,E2 621.4644} C_DIS
LIN {X -135.628,Y -22.8307,Z 161,A -173.3822,B 24.9639,C -1.389,E1 24.8422,E2 620.015} C_DIS
LIN {X -134.9981,Y -26.3037,Z 161,A -171.7257,B 24.9636,C -1.3938,E1 24.8431,E2 618.3374} C_DIS
LIN {X -134.0856,Y -30.6133,Z 161,A -170.0338,B 24.9643,C -1.3806,E1 24.8441,E2 616.6668} C_DIS
LIN {X -133.2435,Y -34.0932,Z 161,A -168.5444,B 24.9645,C -1.3758,E1 24.8451,E2 615.1802} C_DIS
LIN {X -131.9596,Y -38.7656,Z 161,A -165.8957,B 24.9632,C -1.4018,E1 24.8472,E2 612.4541} C_DIS
LIN {X -130.4485,Y -43.581,Z 161,A -164.3611,B 24.965,C -1.3661,E1 24.8485,E2 610.996} C_DIS
LIN {X -129.353,Y -46.7322,Z 161,A -162.9904,B 24.9653,C -1.3609,E1 24.8497,E2 609.6299} C_DIS
LIN {X -128.0872,Y -50.0983,Z 161,A -161.4801,B 24.9655,C -1.357,E1 24.8512,E2 608.1204} C_DIS
LIN {X -126.5574,Y -53.8509,Z 161,A -159.6694,B 24.9655,C -1.3582,E1 24.8532,E2 606.2968} C_DIS
LIN {X -123.2863,Y -60.9636,Z 161,A -156.8784,B 24.9671,C -1.3245,E1 24.8564,E2 603.5706} C_DIS
LIN {X -121.0797,Y -65.2407,Z 161,A -154.3307,B 24.966,C -1.3466,E1 24.8598,E2 600.9567} C_DIS
LIN {X -119.2856,Y -68.4667,Z 161,A -152.8719,B 24.9665,C -1.3383,E1 24.8618,E2 599.5102} C_DIS
LIN {X -117.1052,Y -72.1321,Z 161,A -151.0818,B 24.9667,C -1.3341,E1 24.8644,E2 597.7208} C_DIS
LIN {X -114.7908,Y -75.7608,Z 161,A -148.8378,B 24.9657,C -1.3528,E1 24.8679,E2 595.421} C_DIS
LIN {X -112.2372,Y -79.4952,Z 161,A -147.5365,B 24.9675,C -1.3176,E1 24.8699,E2 594.1972} C_DIS
LIN {X -110.7832,Y -81.5089,Z 161,A -146.2969,B 24.9671,C -1.3256,E1 24.8719,E2 592.9325} C_DIS
LIN {X -107.9604,Y -85.213,Z 161,A -144.3883,B 24.9674,C -1.3191,E1 24.8752,E2 591.0303} C_DIS
LIN {X -105.2518,Y -88.5363,Z 161,A -142.4113,B 24.9671,C -1.3248,E1 24.8788,E2 589.0307} C_DIS
LIN {X -101.8762,Y -92.4004,Z 161,A -140.4056,B 24.9677,C -1.3129,E1 24.8825,E2 587.0443} C_DIS
LIN {X -98.6826,Y -95.8039,Z 161,A -138.3876,B 24.9677,C -1.3124,E1 24.8864,E2 585.0187} C_DIS
LIN {X -95.1502,Y -99.3129,Z 161,A -136.4139,B 24.9682,C -1.3027,E1 24.8903,E2 583.0599} C_DIS
LIN {X -92.0258,Y -102.2153,Z 161,A -133.8267,B 24.9663,C -1.3419,E1 24.8959,E2 580.369} C_DIS
LIN {X -87.1326,Y -106.4167,Z 161,A -132.0475,B 24.9689,C -1.2885,E1 24.8994,E2 578.7101} C_DIS
LIN {X -84.0887,Y -108.8381,Z 161,A -130.1807,B 24.9684,C -1.2985,E1 24.9036,E2 576.8127} C_DIS
LIN {X -80.0761,Y -111.8232,Z 161,A -128.1959,B 24.9689,C -1.2896,E1 24.9081,E2 574.8421} C_DIS
LIN {X -76.5369,Y -114.2748,Z 161,A -126.277,B 24.9687,C -1.2932,E1 24.9125,E2 572.9081} C_DIS
LIN {X -72.2126,Y -117.0558,Z 161,A -124.2724,B 24.9692,C -1.2825,E1 24.9172,E2 570.9225} C_DIS
LIN {X -68.7532,Y -119.1202,Z 161,A -122.5709,B 24.9692,C -1.2813,E1 24.9213,E2 569.2189} C_DIS
LIN {X -65.2602,Y -121.0692,Z 161,A -120.9209,B 24.9694,C -1.2781,E1 24.9254,E2 567.5717} C_DIS
LIN {X -62.0893,Y -122.7236,Z 161,A -119.5074,B 24.9697,C -1.2721,E1 24.9288,E2 566.1686} C_DIS
LIN {X -59.1178,Y -124.182,Z 161,A -118.1036,B 24.9697,C -1.2717,E1 24.9324,E2 564.7622} C_DIS
LIN {X -56.0976,Y -125.5752,Z 161,A -116.4996,B 24.9692,C -1.2818,E1 24.9365,E2 563.1302} C_DIS
LIN {X -52.5198,Y -127.1141,Z 161,A -115.1065,B 24.9699,C -1.2677,E1 24.94,E2 561.7674} C_DIS
LIN {X -49.1974,Y -128.4373,Z 161,A -113.395,B 24.9694,C -1.2782,E1 24.9446,E2 560.0275} C_DIS
LIN {X -45.1029,Y -129.9301,Z 161,A -111.7677,B 24.97,C -1.2664,E1 24.9488,E2 558.4248} C_DIS
LIN {X -41.9341,Y -130.9871,Z 161,A -110.3773,B 24.97,C -1.2652,E1 24.9525,E2 557.0347} C_DIS
LIN {X -38.5712,Y -132.0165,Z 161,A -108.9562,B 24.9702,C -1.2618,E1 24.9563,E2 555.6194} C_DIS
LIN {X -35.2966,Y -132.9296,Z 161,A -107.5164,B 24.9702,C -1.2621,E1 24.9602,E2 554.1765} C_DIS
LIN {X -31.8047,Y -133.8087,Z 161,A -105.8941,B 24.9699,C -1.2679,E1 24.9646,E2 552.5383} C_DIS
LIN {X -26.1488,Y -135.0277,Z 161,A -102.7108,B 24.9679,C -1.3093,E1 24.9736,E2 549.2531} C_DIS
LIN {X -19.7648,Y -136.1088,Z 161,A -101.0901,B 24.9708,C -1.2494,E1 24.9777,E2 547.7731} C_DIS
LIN {X -13.9577,Y -136.8281,Z 161,A -98.338,B 24.97,C -1.2662,E1 24.9854,E2 544.9795} C_DIS
LIN {X -10.8489,Y -137.1095,Z 161,A -97.0957,B 24.9701,C -1.2629,E1 24.9889,E2 543.7444} C_DIS
LIN {X -7.0333,Y -137.3563,Z 161,A -95.5235,B 24.9701,C -1.2619,E1 24.9932,E2 542.1741} C_DIS
LIN {X -0.9045,Y -137.5333,Z 161,A -92.8586,B 24.9699,C -1.2684,E1 25.0007,E2 539.4936} C_DIS
LIN {X -0.9045,Y -137.5333,Z 161,A -92.8586,B 24.9699,C -1.2684,E1 25.0007,E2 539.4936} C_DIS
Enddeposition()
LIN {X 0.9864,Y -136.6083,Z 161,A -93.0585,B 23.0349,C -0.8452,E1 23.0475,E2 540.5038} C_DIS
Startdeposition()
$VEL.CP = VEL_PRINT
LIN {X -5.2784,Y -136.51,Z 161,A -94.5367,B 23.0329,C -0.9015,E1 23.0437,E2 541.8383} C_DIS
LIN {X -12.4231,Y -136.0473,Z 161,A -98.3747,B 23.0344,C -0.8603,E1 23.0327,E2 545.7833} C_DIS
LIN {X -16.9984,Y -135.5521,Z 161,A -99.7275,B 23.0334,C -0.8889,E1 23.0292,E2 547.0639} C_DIS
LIN {X -21.2224,Y -134.9537,Z 161,A -102.5517,B 23.0351,C -0.8391,E1 23.0211,E2 550.0184} C_DIS
LIN {X -28.1681,Y -133.6779,Z 161,A -104.6505,B 23.0336,C -0.8821,E1 23.0156,E2 552.0097} C_DIS
LIN {X -32.4257,Y -132.7083,Z 161,A -106.3417,B 23.0333,C -0.8899,E1 23.011,E2 553.6834} C_DIS
LIN {X -35.6314,Y -131.8838,Z 161,A -107.8819,B 23.0336,C -0.8834,E1 23.0068,E2 555.2428} C_DIS
LIN {X -39.8172,Y -130.6803,Z 161,A -109.6132,B 23.0334,C -0.8893,E1 23.0022,E2 556.962} C_DIS
LIN {X -43.3578,Y -129.5487,Z 161,A -111.1595,B 23.0333,C -0.8912,E1 22.9981,E2 558.5067} C_DIS
LIN {X -46.8519,Y -128.3274,Z 161,A -112.7746,B 23.0333,C -0.8895,E1 22.9938,E2 560.1295} C_DIS
LIN {X -50.7212,Y -126.8472,Z 161,A -114.8424,B 23.0339,C -0.8754,E1 22.9884,E2 562.2385} C_DIS
LIN {X -54.2577,Y -125.3747,Z 161,A -116.084,B 23.0332,C -0.8947,E1 22.9853,E2 563.4338} C_DIS
LIN {X -57.5922,Y -123.8786,Z 161,A -117.5769,B 23.033,C -0.8983,E1 22.9815,E2 564.9214} C_DIS
LIN {X -60.7035,Y -122.384,Z 161,A -119.0312,B 23.033,C -0.8998,E1 22.9779,E2 566.376} C_DIS
LIN {X -64.2123,Y -120.5823,Z 161,A -120.7632,B 23.033,C -0.8982,E1 22.9736,E2 568.1173} C_DIS
LIN {X -68.0711,Y -118.4472,Z 161,A -122.6369,B 23.033,C -0.8997,E1 22.969,E2 569.9932} C_DIS
LIN {X -71.6556,Y -116.3132,Z 161,A -124.6376,B 23.0333,C -0.8904,E1 22.9642,E2 572.0245} C_DIS
LIN {X -74.5822,Y -114.4586,Z 161,A -125.7147,B 23.0326,C -0.9106,E1 22.9617,E2 573.0537} C_DIS
LIN {X -77.5682,Y -112.4566,Z 161,A -127.3585,B 23.0327,C -0.9066,E1 22.9579,E2 574.7138} C_DIS
LIN {X -81.2007,Y -109.8628,Z 161,A -129.4487,B 23.033,C -0.8995,E1 22.9531,E2 576.8302} C_DIS
LIN {X -83.7562,Y -107.9265,Z 161,A -130.5331,B 23.0324,C -0.9143,E1 22.9508,E2 577.8811} C_DIS
LIN {X -91.121,Y -101.785,Z 161,A -134.2422,B 23.0316,C -0.9367,E1 22.943,E2 581.5481} C_DIS
LIN {X -94.6668,Y -98.4964,Z 161,A -136.4775,B 23.0318,C -0.9311,E1 22.9383,E2 583.8078} C_DIS
LIN {X -97.4408,Y -95.7524,Z 161,A -138.1222,B 23.0317,C -0.9342,E1 22.9351,E2 585.4521} C_DIS
LIN {X -99.7108,Y -93.387,Z 161,A -139.7952,B 23.0321,C -0.9233,E1 22.9318,E2 587.1611} C_DIS
LIN {X -104.32,Y -88.2083,Z 161,A -142.4646,B 23.0314,C -0.9411,E1 22.927,E2 589.7979} C_DIS
LIN {X -106.4318,Y -85.6476,Z 161,A -144.0325,B 23.0316,C -0.9363,E1 22.9242,E2 591.3863} C_DIS
LIN {X -109.2916,Y -81.9679,Z 161,A -145.8343,B 23.0311,C -0.9482,E1 22.9211,E2 593.1669} C_DIS
LIN {X -111.4001,Y -79.0786,Z 161,A -147.8761,B 23.032,C -0.9269,E1 22.9177,E2 595.2743} C_DIS
LIN {X -113.7549,Y -75.6512,Z 161,A -149.0836,B 23.0308,C -0.9562,E1 22.9159,E2 596.4132} C_DIS
LIN {X -115.709,Y -72.6277,Z 161,A -150.8002,B 23.031,C -0.9506,E1 22.9133,E2 598.1537} C_DIS
LIN {X -118.0493,Y -68.7585,Z 161,A -152.7108,B 23.0309,C -0.955,E1 22.9106,E2 600.0637} C_DIS
LIN {X -120.6895,Y -64.0081,Z 161,A -154.777,B 23.0302,C -0.9711,E1 22.9079,E2 602.1004} C_DIS
LIN {X -124.8922,Y -55.3609,Z 161,A -158.8604,B 23.0299,C -0.9801,E1 22.903,E2 606.1849} C_DIS
LIN {X -125.9748,Y -52.8497,Z 161,A -160.1477,B 23.0299,C -0.977,E1 22.9015,E2 607.4882} C_DIS
LIN {X -127.3618,Y -49.4135,Z 161,A -161.6502,B 23.0297,C -0.984,E1 22.9,E2 608.9819} C_DIS
LIN {X -128.6078,Y -46.0741,Z 161,A -163.1816,B 23.0297,C -0.9867,E1 22.8985,E2 610.5157} C_DIS
LIN {X -129.9768,Y -42.0596,Z 161,A -165.0064,B 23.0295,C -0.99,E1 22.8969,E2 612.3436} C_DIS
LIN {X -132.0367,Y -35.0583,Z 161,A -168.0624,B 23.0291,C -0.9996,E1 22.8945,E2 615.3943} C_DIS
LIN {X -133.0569,Y -30.9667,Z 161,A -170.2892,B 23.0297,C -0.9842,E1 22.893,E2 617.6749} C_DIS
LIN {X -133.9307,Y -26.9337,Z 161,A -171.5241,B 23.0286,C -1.0122,E1 22.8924,E2 618.8459} C_DIS
LIN {X -134.5014,Y -23.9203,Z 161,A -172.8742,B 23.0286,C -1.0134,E1 22.8917,E2 620.2017} C_DIS
LIN {X -135.1716,Y -19.7899,Z 161,A -174.7248,B 23.0285,C -1.0146,E1 22.8909,E2 622.0612} C_DIS
LIN {X -135.7033,Y -15.7358,Z 161,A -176.4764,B 23.0283,C -1.0184,E1 22.8903,E2 623.8146} C_DIS
LIN {X -136.1243,Y -11.5324,Z 161,A -178.1614,B 23.0279,C -1.028,E1 22.8899,E2 625.4858} C_DIS
LIN {X -136.3927,Y -7.7623,Z 161,A -179.8068,B 23.0278,C -1.0304,E1 22.8896,E2 627.136} C_DIS
LIN {X -136.5593,Y -3.795,Z 161,A 178.5439,B 23.0275,C -1.0365,E1 22.8894,E2 628.7804} C_DIS
LIN {X -136.613,Y 0.2913,Z 161,A 176.7692,B 23.0275,C -1.0393,E1 22.8894,E2 630.5597} C_DIS
LIN {X -136.5498,Y 4.1352,Z 161,A 175.2222,B 23.0271,C -1.0476,E1 22.8894,E2 632.0957} C_DIS
LIN {X -136.3692,Y 8.1438,Z 161,A 173.472,B 23.027,C -1.05,E1 22.8897,E2 633.8512} C_DIS
LIN {X -136.0434,Y 12.4638,Z 161,A 171.5797,B 23.0269,C -1.0525,E1 22.8902,E2 635.7496} C_DIS
LIN {X -135.6181,Y 16.4499,Z 161,A 169.9486,B 23.0265,C -1.0602,E1 22.8907,E2 637.3714} C_DIS
LIN {X -135.0346,Y 20.7001,Z 161,A 168.1651,B 23.0262,C -1.0668,E1 22.8914,E2 639.1498} C_DIS
LIN {X -134.4857,Y 24.0076,Z 161,A 166.779,B 23.026,C -1.0722,E1 22.892,E2 640.5308} C_DIS
LIN {X -133.8333,Y 27.4124,Z 161,A 165.3294,B 23.0258,C -1.0771,E1 22.8928,E2 641.9773} C_DIS
LIN {X -133.1189,Y 30.6953,Z 161,A 163.9063,B 23.0256,C -1.081,E1 22.8937,E2 643.3995} C_DIS
LIN {X -132.3405,Y 33.8947,Z 161,A 162.5193,B 23.0254,C -1.0851,E1 22.8946,E2 644.7848} C_DIS
LIN {X -131.4708,Y 37.1253,Z 161,A 161.0937,B 23.0253,C -1.0886,E1 22.8957,E2 646.2106} C_DIS
LIN {X -130.3441,Y 40.91,Z 161,A 159.395,B 23.0251,C -1.0919,E1 22.8971,E2 647.9116} C_DIS
LIN {X -129.0788,Y 44.7369,Z 161,A 157.6576,B 23.025,C -1.0951,E1 22.8986,E2 649.6516} C_DIS
LIN {X -127.726,Y 48.4678,Z 161,A 156.075,B 23.0246,C -1.1039,E1 22.9002,E2 651.2212} C_DIS
LIN {X -126.6425,Y 51.2291,Z 161,A 154.7918,B 23.0245,C -1.106,E1 22.9015,E2 652.5069} C_DIS
LIN {X -125.2253,Y 54.603,Z 161,A 153.2585,B 23.0243,C -1.1108,E1 22.9032,E2 654.0373} C_DIS
LIN {X -123.7444,Y 57.8824,Z 161,A 151.5629,B 23.0244,C -1.1068,E1 22.9052,E2 655.7531} C_DIS
LIN {X -121.3438,Y 62.762,Z 161,A 149.0328,B 23.0246,C -1.1023,E1 22.9084,E2 658.3097} C_DIS
LIN {X -119.5598,Y 66.0962,Z 161,A 147.7366,B 23.0238,C -1.1201,E1 22.9101,E2 659.5676} C_DIS
LIN {X -117.2092,Y 70.1805,Z 161,A 145.7479,B 23.0236,C -1.1253,E1 22.9129,E2 661.5544} C_DIS
LIN {X -114.9248,Y 73.862,Z 161,A 143.5129,B 23.0242,C -1.1115,E1 22.9163,E2 663.8372} C_DIS
LIN {X -112.4982,Y 77.5077,Z 161,A 142.0699,B 23.0232,C -1.1345,E1 22.9185,E2 665.229} C_DIS
LIN {X -109.8433,Y 81.2272,Z 161,A 139.8146,B 23.0236,C -1.1243,E1 22.9223,E2 667.5225} C_DIS
LIN {X -107.4698,Y 84.3414,Z 161,A 138.7624,B 23.0222,C -1.1556,E1 22.924,E2 668.4996} C_DIS
LIN {X -104.6177,Y 87.8542,Z 161,A 136.7875,B 23.0222,C -1.157,E1 22.9275,E2 670.481} C_DIS
LIN {X -103.0614,Y 89.675,Z 161,A 135.578,B 23.0224,C -1.1502,E1 22.9297,E2 671.714} C_DIS
LIN {X -100.0757,Y 92.9951,Z 161,A 133.6796,B 23.0223,C -1.1538,E1 22.9333,E2 673.6125} C_DIS
LIN {X -96.8908,Y 96.3089,Z 161,A 131.742,B 23.0221,C -1.158,E1 22.9371,E2 675.5482} C_DIS
LIN {X -93.6619,Y 99.4519,Z 161,A 129.8472,B 23.0219,C -1.1623,E1 22.9409,E2 677.4407} C_DIS
LIN {X -90.2943,Y 102.5194,Z 161,A 127.9666,B 23.0216,C -1.1681,E1 22.9448,E2 679.3147} C_DIS
LIN {X -86.9313,Y 105.3861,Z 161,A 126.1005,B 23.0214,C -1.1716,E1 22.9488,E2 681.1795} C_DIS
LIN {X -83.2681,Y 108.3041,Z 161,A 124.2072,B 23.021,C -1.1791,E1 22.9529,E2 683.0613} C_DIS
LIN {X -80.4026,Y 110.4479,Z 161,A 122.5825,B 23.0212,C -1.1765,E1 22.9566,E2 684.699} C_DIS
LIN {X -76.6024,Y 113.1163,Z 161,A 120.8608,B 23.0205,C -1.1909,E1 22.9604,E2 686.3901} C_DIS
LIN {X -72.091,Y 116.0436,Z 161,A 118.3966,B 23.0207,C -1.1854,E1 22.9663,E2 688.8771} C_DIS
LIN {X -68.5507,Y 118.1696,Z 161,A 115.9354,B 23.0222,C -1.1547,E1 22.9725,E2 691.425} C_DIS
LIN {X -63.4908,Y 120.9611,Z 161,A 114.6121,B 23.0195,C -1.2101,E1 22.9754,E2 692.6104} C_DIS
LIN {X -59.7246,Y 122.8669,Z 161,A 112.5166,B 23.0201,C -1.1976,E1 22.9807,E2 694.7441} C_DIS
LIN {X -57.0807,Y 124.1151,Z 161,A 111.2715,B 23.0201,C -1.1986,E1 22.9838,E2 695.99} C_DIS
LIN {X -54.0547,Y 125.4624,Z 161,A 109.8992,B 23.02,C -1.2015,E1 22.9873,E2 697.3585} C_DIS
LIN {X -47.5575,Y 128.067,Z 161,A 106.9281,B 23.0198,C -1.2037,E1 22.9951,E2 700.3309} C_DIS
LIN {X -41.7246,Y 130.0839,Z 161,A 103.7663,B 23.021,C -1.1798,E1 23.0036,E2 703.5604} C_DIS
LIN {X -37.1255,Y 131.4708,Z 161,A 102.5125,B 23.0191,C -1.218,E1 23.0067,E2 704.7187} C_DIS
LIN {X -33.4052,Y 132.4647,Z 161,A 100.685,B 23.0196,C -1.2094,E1 23.0117,E2 706.571} C_DIS
LIN {X -29.4333,Y 133.4047,Z 161,A 98.8987,B 23.0196,C -1.2074,E1 23.0166,E2 708.365} C_DIS
LIN {X -25.6804,Y 134.1763,Z 161,A 97.3318,B 23.0195,C -1.2106,E1 23.0209,E2 709.9256} C_DIS
LIN {X -22.3091,Y 134.778,Z 161,A 95.9474,B 23.0193,C -1.2142,E1 23.0247,E2 711.3025} C_DIS
LIN {X -18.6814,Y 135.33,Z 161,A 94.2675,B 23.0196,C -1.2084,E1 23.0294,E2 712.9987} C_DIS
LIN {X -12.8375,Y 136.0076,Z 161,A 91.8868,B 23.0193,C -1.2138,E1 23.0359,E2 715.367} C_DIS
LIN {X -8.5526,Y 136.3441,Z 161,A 90.0806,B 23.0193,C -1.2144,E1 23.041,E2 717.1725} C_DIS
LIN {X -3.0604,Y 136.5796,Z 161,A 87.3333,B 23.0203,C -1.1938,E1 23.0488,E2 719.973} C_DIS
LIN {X 1.15,Y 136.6078,Z 161,A 86.0706,B 23.0191,C -1.2184,E1 23.0521,E2 721.1727} C_DIS
LIN {X 5.1776,Y 136.5139,Z 161,A 83.8377,B 23.0204,C -1.1922,E1 23.0585,E2 723.4719} C_DIS
LIN {X 9.6804,Y 136.2688,Z 161,A 82.1036,B 23.02,C -1.1997,E1 23.0633,E2 725.186} C_DIS
LIN {X 13.3253,Y 135.9607,Z 161,A 80.9773,B 23.0191,C -1.2193,E1 23.0663,E2 726.2614} C_DIS
LIN {X 16.6088,Y 135.5992,Z 161,A 79.4166,B 23.0195,C -1.2105,E1 23.0707,E2 727.8434} C_DIS
LIN {X 25.1872,Y 134.2706,Z 161,A 76.0526,B 23.0189,C -1.2228,E1 23.0799,E2 731.1723} C_DIS
LIN {X 28.7926,Y 133.5431,Z 161,A 74.3826,B 23.0192,C -1.2158,E1 23.0845,E2 732.8579} C_DIS
LIN {X 31.834,Y 132.851,Z 161,A 73.0394,B 23.0194,C -1.2133,E1 23.0881,E2 734.2054} C_DIS
LIN {X 35.3624,Y 131.9556,Z 161,A 71.5308,B 23.0194,C -1.2133,E1 23.0922,E2 735.7116} C_DIS
LIN {X 38.8121,Y 130.983,Z 161,A 70.0324,B 23.0194,C -1.2124,E1 23.0962,E2 737.2095} C_DIS
LIN {X 42.1835,Y 129.9373,Z 161,A 68.56,B 23.0194,C -1.2115,E1 23.1001,E2 738.681} C_DIS
LIN {X 45.9684,Y 128.6459,Z 161,A 67.0593,B 23.0191,C -1.2188,E1 23.1041,E2 740.1599} C_DIS
LIN {X 52.2326,Y 126.2325,Z 161,A 64.1017,B 23.0196,C -1.2089,E1 23.1118,E2 743.1356} C_DIS
LIN {X 56.017,Y 124.5988,Z 161,A 62.4189,B 23.0196,C -1.2092,E1 23.1161,E2 744.8131} C_DIS
LIN {X 58.9039,Y 123.26,Z 161,A 60.9922,B 23.0199,C -1.203,E1 23.1197,E2 746.2518} C_DIS
LIN {X 62.3422,Y 121.5578,Z 161,A 59.4264,B 23.0199,C -1.203,E1 23.1236,E2 747.8127} C_DIS
LIN {X 65.3089,Y 119.9917,Z 161,A 57.9131,B 23.0202,C -1.1957,E1 23.1274,E2 749.3399} C_DIS
LIN {X 69.3805,Y 117.6844,Z 161,A 55.9632,B 23.0203,C -1.1935,E1 23.1321,E2 751.289} C_DIS
LIN {X 73.1536,Y 115.377,Z 161,A 54.1094,B 23.0205,C -1.1906,E1 23.1365,E2 753.1436} C_DIS
LIN {X 76.9372,Y 112.8897,Z 161,A 52.2081,B 23.0206,C -1.1874,E1 23.1409,E2 755.0463} C_DIS
LIN {X 80.7029,Y 110.2285,Z 161,A 50.4562,B 23.0204,C -1.1932,E1 23.1448,E2 756.7765} C_DIS
LIN {X 83.4657,Y 108.1517,Z 161,A 48.1799,B 23.0225,C -1.1488,E1 23.1501,E2 759.1568} C_DIS
LIN {X 87.9786,Y 104.5122,Z 161,A 46.5842,B 23.0207,C -1.1864,E1 23.1533,E2 760.6501} C_DIS
LIN {X 90.278,Y 102.5338,Z 161,A 45.188,B 23.0211,C -1.1775,E1 23.1563,E2 762.063} C_DIS
LIN {X 93.4875,Y 99.6165,Z 161,A 43.2948,B 23.0215,C -1.1699,E1 23.1602,E2 763.9669} C_DIS
LIN {X 96.1131,Y 97.0853,Z 161,A 41.8917,B 23.0213,C -1.1731,E1 23.163,E2 765.3556} C_DIS
LIN {X 99.0774,Y 94.0589,Z 161,A 40.0863,B 23.0216,C -1.1677,E1 23.1665,E2 767.1661} C_DIS
LIN {X 102.2712,Y 90.5751,Z 161,A 38.2961,B 23.0213,C -1.1731,E1 23.1698,E2 768.9341} C_DIS
LIN {X 104.465,Y 88.0362,Z 161,A 36.6862,B 23.022,C -1.1593,E1 23.1727,E2 770.5709} C_DIS
LIN {X 107.2967,Y 84.5618,Z 161,A 34.9106,B 23.022,C -1.1601,E1 23.1758,E2 772.3353} C_DIS
LIN {X 109.562,Y 81.6051,Z 161,A 32.9166,B 23.0232,C -1.134,E1 23.1793,E2 774.3852} C_DIS
LIN {X 111.9721,Y 78.2652,Z 161,A 31.7134,B 23.0221,C -1.1566,E1 23.1811,E2 775.5246} C_DIS
LIN {X 113.4564,Y 76.0984,Z 161,A 30.4457,B 23.0227,C -1.1452,E1 23.1831,E2 776.8146} C_DIS
LIN {X 115.8478,Y 72.4057,Z 161,A 28.6115,B 23.0229,C -1.1409,E1 23.1859,E2 778.6496} C_DIS
LIN {X 118.0727,Y 68.718,Z 161,A 26.8278,B 23.023,C -1.1371,E1 23.1884,E2 780.4327} C_DIS
LIN {X 120.204,Y 64.9178,Z 161,A 25.034,B 23.0232,C -1.1338,E1 23.1908,E2 782.2247} C_DIS
LIN {X 121.7932,Y 61.8797,Z 161,A 23.6368,B 23.0232,C -1.132,E1 23.1926,E2 783.6185} C_DIS
LIN {X 123.4784,Y 58.4466,Z 161,A 22.0991,B 23.0233,C -1.1308,E1 23.1945,E2 785.1501} C_DIS
LIN {X 124.9551,Y 55.2204,Z 161,A 20.4951,B 23.0238,C -1.1205,E1 23.1963,E2 786.7708} C_DIS
LIN {X 126.5486,Y 51.462,Z 161,A 18.7747,B 23.0241,C -1.115,E1 23.1982,E2 788.4946} C_DIS
LIN {X 127.9924,Y 47.7567,Z 161,A 17.2253,B 23.0241,C -1.1163,E1 23.1997,E2 790.0315} C_DIS
LIN {X 130.5903,Y 40.1114,Z 161,A 13.8722,B 23.0244,C -1.1077,E1 23.2027,E2 793.3855} C_DIS
LIN {X 131.5885,Y 36.7046,Z 161,A 12.401,B 23.0246,C -1.1041,E1 23.2038,E2 794.8568} C_DIS
LIN {X 132.4885,Y 33.3114,Z 161,A 10.941,B 23.0247,C -1.1002,E1 23.2048,E2 796.3175} C_DIS
LIN {X 133.3566,Y 29.6544,Z 161,A 9.3541,B 23.025,C -1.0946,E1 23.2058,E2 797.9084} C_DIS
LIN {X 134.1538,Y 25.7981,Z 161,A 7.7227,B 23.0252,C -1.0905,E1 23.2067,E2 799.5398} C_DIS
LIN {X 134.7547,Y 22.4489,Z 161,A 6.3047,B 23.0254,C -1.0865,E1 23.2074,E2 800.959} C_DIS
LIN {X 135.3483,Y 18.5531,Z 161,A 4.7156,B 23.0254,C -1.0845,E1 23.208,E2 802.5429} C_DIS
LIN {X 135.8708,Y 14.2162,Z 161,A 2.8588,B 23.0258,C -1.0773,E1 23.2086,E2 804.4058} C_DIS
Enddeposition()
END
